ACTION Control:
IF NOT bRUN THEN
				lrGearRatio:=-ABS(lrLifterStopDosePosition-lrLifterStartDosePosition+0.000000000001)
							/(*---------------------------------------------------------------------*)
							((BOOL_TO_INT(bLiftSynchroPh1)*lrDosePhase1Volume)
							+(BOOL_TO_INT(bLiftSynchroPh2)*(lrDoseVolume-lrDosePhase2Volume-lrDosePhase1Volume))
							+((BOOL_TO_INT(bLiftSynchroPh3)*(lrDoseVolume-lrDosePhase1Volume)))
							+ 0.000000000001); 					
	drugafaza:=(lrDoseVolume-lrDosePhase2Volume-lrDosePhase1Volume);						
	trzeciafaza:=(lrDoseVolume-lrDosePhase2Volume);
	calosc:=(*---------------------------------------------------------------------*)
							((BOOL_TO_INT(bLiftSynchroPh1)*lrDosePhase1Volume)
							+(BOOL_TO_INT(bLiftSynchroPh2)*(lrDoseVolume-lrDosePhase2Volume-lrDosePhase1Volume))
							+((BOOL_TO_INT(bLiftSynchroPh3)*lrDosePhase2Volume))
							+ 0.000000000001);
END_IF
	



	(** TIMERY**)
	tonDoseValveOpenTimeAcc(	IN:= eRunningState = E_DispencerState.eDosingPh1, 											PT:= LREAL_TO_TIME(lrDoseValveOpenTimeAcc));   		// [1] Przyśpieszenie otwarcia zaworu tłoczenia [ms]
	tonDoseValveCloseTimeDec(	IN:= (eRunningState=E_DispencerState.eDosingPh3 AND NOT bDoseSucking) OR
									 (eRunningState=E_DispencerState.eDoseSucking AND mcDispencerMoveAbsolute1.Done),		PT:= LREAL_TO_TIME(lrDoseValveCloseTimeDec));  		// [2] Opóźnienie zamknięcia zaworu tłoczenia [ms]
	tonSuckValveOpenTimeDelay(	IN:= eRunningState = E_DispencerState.eGoingUp,											PT:= LREAL_TO_TIME(lrSuckValveOpenTimeDelay));		// [3] Opóżnienie rozpoczęcia ssania po tłoczeniu [ms]
	tonSuckValveCloseTimeDelay(	IN:= (eRunningState = E_DispencerState.eSucking OR 
										eRunningState = E_DispencerState.eDosingDone											
																	) AND
										 mcDispencerMoveAbsolute1.Done, 												PT:= LREAL_TO_TIME(lrSuckValveCloseTimeDelay)); 	// [4] Opóżnienie zamknięcia zaworu ssącego [ms]
	tonDoseSuckingTimeDelay(	IN:= eRunningState = E_DispencerState.eDoseSucking,										PT:= LREAL_TO_TIME(lrDoseSuckingTimeDelay));    	// [6] [Podsysanie] Opóźnienie podsysania [ms]

	//Opóźnienie potwierdzenia wykonania dozy
	(*tonDosingDoneDelay(IN:=(eRunningState=E_DispencerState.eDosingDone OR eRunningState=E_DispencerState.eSucking)AND
							mcDispencerMoveAbsolute1.Done AND tonSuckValveCloseTimeDelay.Q 				
							, PT:=UDINT_TO_TIME(nDosingDoneDelayTime));*)
	tonPrepareToAborting(IN:=bPrepareToAborting, PT:=T#1S);
	//Opóźnienie potwierdzenia wykonania dozy Zmiana 20200820
	tonDosingDoneDelay(IN:=(eRunningState=E_DispencerState.eDosingDone OR eRunningState=E_DispencerState.eSucking)				
							, PT:=UDINT_TO_TIME(nDosingDoneDelayTime));
							
	tonDelayServoOn(IN:=(eState = E_Station.ePreparingToReady), PT:=T#7S); ////bylo 3 Nowe XTS bylo 1200ms						
	tonDelayEnable(IN:=	bEnable, PT:=T#5S);			
	(*Synchronizacja tylko jedna zaznaczona*)
	(*Zabezpieczenie przed zalaczeniem trzech*)
(*	rtLiftSynchroPh3(CLK:=bLiftSynchroPh3,Q=>);rtLiftSynchroPh2(CLK:=bLiftSynchroPh2,Q=>);rtLiftSynchroPh1(CLK:=bLiftSynchroPh1,Q=>);
	IF rtLiftSynchroPh1.Q THEN	bLiftSynchroPh2:=FALSE;	bLiftSynchroPh3:=FALSE; END_IF
	IF rtLiftSynchroPh2.Q THEN	bLiftSynchroPh1:=FALSE;	bLiftSynchroPh3:=FALSE; END_IF
	IF rtLiftSynchroPh3.Q THEN	bLiftSynchroPh1:=FALSE;	bLiftSynchroPh2:=FALSE; END_IF 
	IF bLiftSynchroPh1 THEN	bLiftSynchroPh2:=FALSE;	bLiftSynchroPh3:=FALSE;
	ELSIF bLiftSynchroPh2 THEN	bLiftSynchroPh1:=FALSE;	bLiftSynchroPh3:=FALSE;
	ELSIF bLiftSynchroPh3 THEN	bLiftSynchroPh1:=FALSE;	bLiftSynchroPh2:=FALSE;
	ELSIF NOT bLiftSynchroPh1  AND NOT bLiftSynchroPh2 AND NOT bLiftSynchroPh3 THEN	bLiftSynchroPh1:=TRUE;	bLiftSynchroPh2:=FALSE;	bLiftSynchroPh3:=FALSE; END_IF
	(*Koniec Zabezpieczenie przed zalaczeniem trzech*)
*)
	
	//	100					300			250
	IF lrDosePhase1Volume>lrDoseVolume-lrDosePhase2Volume THEN
		lrDosePhase1Volume:=lrDoseVolume-lrDosePhase2Volume;
	END_IF
	// 200					300			200
	IF lrDosePhase2Volume>lrDoseVolume-lrDosePhase1Volume THEN
		lrDosePhase2Volume:=lrDoseVolume-lrDosePhase1Volume;
	END_IF
	
	IF  eState=E_Station.eReady OR eRunningState=E_DispencerState.eDosingDone OR eRunningState=E_DispencerState.eGoingUp THEN
//	IF  (eState>E_Station.eError AND eState<=E_Station.eReady) OR eRunningState=E_DispencerState.eDosingDone OR eRunningState=E_DispencerState.eGoingUp THEN
		IF (DispencerLifterAxisRef.NcToPlc.ActPos  >= lrDropCatcherHeightCV+(lrDropCatcherOpenDistance-5)) AND lrDropCatcherHeightCV>1 AND NOT bHoming AND NOT bHeightSet THEN
			bDropCatcherActuator:=TRUE;
		ELSE
			bDropCatcherActuator:=FALSE;
		END_IF
	END_IF
							
							
	//Zbocza 
	rtDosingPh1(CLK:=eRunningState=E_DispencerState.eDosingPh1,Q=>);
	rtDosingPh2(CLK:=eRunningState=E_DispencerState.eDosingPh2,Q=>);
	rtDosingPh3(CLK:=eRunningState=E_DispencerState.eDosingPh3,Q=>);
	rtGoingUp(CLK:=eRunningState=E_DispencerState.eGoingUp,Q=>);
	rtPreparingToDose(CLK:=eRunningState=E_DispencerState.ePreparingToDose,Q=>);	
	
	(*****Wyłączenie enable*****)
	IF NOT bEnable THEN
		IF eState <> E_Station.eDisabled AND eState <> E_Station.ePreparingToDisable THEN
				eState 				:= E_Station.ePreparingToDisable; 
				bCycleDone			:= FALSE;
		END_IF	
	END_IF

	(*****Estop*****)
	IF (NOT bEstop AND bInLimitSwitchSensor) OR (NOT bEStopButtonsAndDoors AND NOT bInLimitSwitchSensor) THEN	
		IF eState <> E_Station.eAborted AND eState <> E_Station.eAborting AND eState <> E_Station.eDisabled THEN
				eState 				:= E_Station.eAborting; 
		END_IF
	END_IF

	
	CASE eState OF
	/////////////////////////////	
		E_Station.eDisabled: 					// Stan nieaktywnosci (Stacja wyłączona) 
		
			IF bEnable AND tonDelayEnable.Q THEN
				eState 				:= E_Station.ePreparingToReady; 
			END_IF 
			
    /////////////////////////////	    
		E_Station.eAborted: 					// Stan bezpiecznego zatrzymania (po Abortingu) 

			IF bEStop THEN
				eState 				:= E_Station.ePreparingToReady;
			END_IF
			
	/////////////////////////////	
		E_Station.eAborting:                 	// Stan bezpiecznego zatrzymywania (po EStopie)
		
			mcDispencerPower.Override			:= 100;
			mcDispencerStop.Execute				:= NOT bStopped AND bDispencerServoPower; //Nowe XTS
			mcDispencerMoveAbsolute1.Execute	:= FALSE;
			mcDispencerMoveAbsolute2.Execute	:= FALSE;
			mcDispencerManualMove.JogBackwards	:= FALSE;
			mcDispencerManualMove.JogForward	:= FALSE;			
			
			IF bDispencerWithLifter THEN (*n*)
				mcLifterPower.Override				:= 100;
				mcLifterStop.Execute				:= NOT bStopped AND bLifterServoPower; //Nowe XTS
				mcLifterMoveAbsolute.Execute		:= FALSE;	
				mcLifterManualMove.JogBackwards		:= FALSE;
				mcLifterManualMove.JogForward		:= FALSE;
				bHeightSetNotDone 					:= FALSE; //Zmiana 2021-02-19
			END_IF	
											(*n*)					//Zmiana XTS
			IF ((mcLifterStop.Done OR NOT bDispencerWithLifter OR NOT bLifterServoPower) AND (mcDispencerStop.Done OR NOT bDispencerServoPower)) OR bStopped THEN
				
				mcDispencerStop.Execute			:=	FALSE;
				bDispencerServoPower			:=	FALSE;
				
				mcLifterStop.Execute			:=	FALSE;
				bLifterServoPower				:=	FALSE;
				
				bStopped						:=	FALSE;
				eState							:=	E_Station.eAborted; 
				eRunningState					:=	E_DispencerState.eReady;
			END_IF	
					
	/////////////////////////////			
		E_Station.eError:                 	 	// Stan błędu 	
			
			IF bReset OR tofReset.Q THEN
				eState 				:= E_Station.eResetting;
				eRunningState		:= E_DispencerState.eReady;
			ELSE
				mcLifterSoftReset	(Execute:=FALSE,Axis:=DispencerLifterAxisRef);
				mcDispencerSoftReset(Execute:=FALSE,Axis:=DispencerAxisRef);
			END_IF
			
	/////////////////////////////
		E_Station.eResetting:					// Stan resetowania bledu (po Errorze)
			
			//Procedura obsługi resetu w zależności od błędu
			CASE nErrorNr-iStationIndex OF
		
				//Error 2 - BŁĄD SERWA DOZOWNIKA
				1:	
					mcDispencerSoftReset(Execute:=TRUE,Axis:=DispencerAxisRef);
					IF mcLifterGearIn.InGear THEN
						mcLifterGearIn.Enable:=FALSE;
						mcLifterGearOut.Execute := TRUE;
					END_IF
					IF mcLifterGearOut.Done THEN
						mcLifterGearOut.Execute := FALSE;
					END_IF
					IF NOT mcLifterGearIn.InGear AND NOT mcLifterGearOut.Execute THEN
					
						IF NOT fbDispencerHardReset.Busy AND NOT mcDispencerSoftReset.Busy AND mcDispencerPower.Status AND NOT DispencerAxisRef.Status.Error THEN
								mcDispencerSoftReset(Execute:=FALSE,Axis:=DispencerAxisRef);
								nErrorNr:=0;
								nDispencerServoErrorNr:=0;
								bError := FALSE;
								sErrorDescription:='';	
				
						ELSIF NOT fbDispencerHardReset.Busy AND NOT mcDispencerSoftReset.Busy AND NOT mcDispencerPower.Status AND NOT DispencerAxisRef.Status.Error THEN
								nErrorNr:=0;
								nDispencerServoErrorNr:=0;
								bError := FALSE;
								sErrorDescription:='';
						END_IF
						IF fbDispencerHardReset.Error OR mcDispencerSoftReset.Error THEN
							mcDispencerSoftReset(Execute:=FALSE,Axis:=DispencerAxisRef);
						END_IF
						
					END_IF

				//Error 2, Error 4 - BŁĄD SERWA PODNOSZENIA DOZOWNIKA
				2:	
					mcLifterGearIn.Enable:=FALSE;
					mcLifterGearOut.Execute:=FALSE;
					//fbLifterHardReset(Execute:=NOT mcLifterMoveAbsolute.Execute,Axis:=DispencerLifterAxisRef);
					mcLifterSoftReset(Execute:=NOT mcLifterMoveAbsolute.Execute,Axis:=DispencerLifterAxisRef);
					IF NOT fbLifterHardReset.Busy AND NOT mcLifterSoftReset.Busy AND mcLifterPower.Status AND NOT DispencerLifterAxisRef.Status.Error THEN
						//fbLifterHardReset(Execute:=FALSE,Axis:=DispencerLifterAxisRef);
						mcLifterSoftReset(Execute:=FALSE,Axis:=DispencerLifterAxisRef);
						mcLifterMoveAbsolute.Execute:=TRUE;
						mcLifterMoveAbsolute.Position:=lrLifterReadyPosition;
						mcLifterPower.Override:=100; 
						IF mcLifterMoveAbsolute.Done THEN
							bDropCatcherActuator:=TRUE;
							mcLifterPower.Override:=100; 
							mcLifterMoveAbsolute.Execute:=FALSE;
							nErrorNr:=0;
							nLifterServoErrorNr:=0;
							bError := FALSE;
							sErrorDescription:='';	
						END_IF 
					ELSIF NOT fbLifterHardReset.Busy AND NOT mcLifterSoftReset.Busy AND NOT mcLifterPower.Status AND NOT DispencerLifterAxisRef.Status.Error THEN		
						//fbLifterHardReset(Execute:=FALSE,Axis:=DispencerLifterAxisRef);
						mcLifterSoftReset(Execute:=FALSE,Axis:=DispencerLifterAxisRef);
						nErrorNr:=0;
						nLifterServoErrorNr:=0;
						bError := FALSE;
						sErrorDescription:='';	
					END_IF
					IF fbLifterHardReset.Error OR mcLifterSoftReset.Error THEN
						//fbLifterHardReset(Execute:=FALSE,Axis:=DispencerLifterAxisRef);
						mcLifterSoftReset(Execute:=FALSE,Axis:=DispencerLifterAxisRef);
					END_IF	

				// inny numer błędu
				ELSE
					bSuckingValveActuator:=FALSE;
					bDosingValveActuator:=FALSE;
					IF bDispencerWithLifter THEN
						mcLifterSoftReset(Execute:=FALSE,Axis:=DispencerLifterAxisRef);
						mcLifterPower.Override				:=	100; 
						mcLifterMoveAbsolute.Acceleration	:=	lrLifterAcceleration;
						mcLifterMoveAbsolute.Velocity		:=	lrLifterVelocity;
						mcLifterMoveAbsolute.Position		:=	lrLifterReadyPosition;
						mcLifterMoveAbsolute.Execute		:=	bLifterServoPower; 
						IF mcLifterMoveAbsolute.Done OR NOT bLifterServoPower THEN 
							bDropCatcherActuator:=TRUE;
							mcLifterPower.Override:=100; 
							mcLifterMoveAbsolute.Execute:=FALSE;
							nErrorNr:=0;
							nLifterServoErrorNr:=0;
							bError := FALSE;
							sErrorDescription:='';	
						END_IF
					ELSE
						bError := FALSE;
					END_IF 

			END_CASE	
			
			IF NOT bError THEN
				nErrorNr 			:=	0;
   				sErrorDescription 	:=	'';
	
				eState 				:=	E_Station.ePreparingToReady;
			ELSE
				eState 				:=	E_Station.eError;
			END_IF
        
	/////////////////////////////
		E_Station.eManualMovement:     			// Stan ruchów manualnych  
       
			ManualMovements();
			//Wyjście z trybu serwisowego
			IF NOT bManualMovement AND bInLimitSwitchSensor  AND NOT bChangeover THEN
				mcDispencerPower.Override			:=	100;		
				bSuckingValveActuator				:=	FALSE;
				bDosingValveActuator				:=	FALSE;
				mcDispencerMoveAbsolute1.Execute	:=	FALSE;
			
				IF bDispencerWithLifter THEN
					IF lrLifterActualPosition < lrLifterReadyPosition + 1 THEN
						mcLifterMoveAbsolute.Execute		:= TRUE;
						mcLifterMoveAbsolute.Acceleration	:= lrLifterAcceleration;
						mcLifterMoveAbsolute.Velocity		:= lrLifterVelocity;
						mcLifterMoveAbsolute.Position		:= lrLifterReadyPosition;
					END_IF
				END_IF
				
				IF NOT bDispencerWithLifter OR mcLifterMoveAbsolute.Done OR lrLifterActualPosition >= lrLifterReadyPosition THEN
					mcDispencerMoveAbsolute1.Execute:=FALSE;
					mcLifterMoveAbsolute.Execute:=FALSE;
					eState 							:= E_Station.eReady;
				END_IF
			END_IF

	/////////////////////////////
		E_Station.eHoming:						// Stan bazowania 

			Homing();
			IF NOT bHoming AND NOT bHeightSet THEN
			   eState:=E_Station.ePreparingToReady;
			   	mcLifterManualMove.JogForward		:= FALSE;
				mcLifterManualMove.JogBackwards		:= FALSE;
			END_IF			
			
	/////////////////////////////
		E_Station.eHomingDone:                  // Stan wykonania bazowania 
		
			bHomingDone							:=	TRUE;
			IF NOT bHoming AND NOT bHeightSet THEN
				
			   eState:=E_Station.eReady;
			END_IF
			
	/////////////////////////////
		E_Station.ePreparingToReady:            // Stan przygotowywania do gotowosci (zawsze przed Ready)  

		
			IF tonDelayServoOn.Q THEN
				bDispencerServoPower		:= TRUE;		
				bLifterServoPower			:= TRUE;//bDispencerWithLifter	; (*n*) //ZMIANA XTS
			END_IF	
		
			mcDispencerPower.Override	:= 100;
			bDosingValveActuator		:= FALSE;
			bSuckingValveActuator		:= FALSE;
			bManualDosingValve			:= FALSE;
			bManualSuckingValve			:= FALSE;
			bServiceBrakeOff			:= FALSE;

			mcLifterMoveAbsolute.Execute := FALSE;

			mcDispencerMoveAbsolute1.Execute := FALSE;
			mcDispencerMoveAbsolute2.Execute := FALSE;
			mcDispencerMoveAbsolute3.Execute := FALSE;
				(*n*)
			IF (mcLifterPower.Status OR NOT bDispencerWithLifter) AND mcDispencerPower.Status THEN
											(*n*)
				IF NOT bHeightSetNotDone AND bDispencerWithLifter THEN
					
					IF mcLifterGearIn.InGear THEN
						mcLifterGearIn.Enable := FALSE;
						mcLifterGearOut.Execute := TRUE;
					ELSIF mcLifterGearIn.Enable AND mcLifterGearOut.Done THEN 
						mcLifterGearOut.Execute := FALSE;
					ELSE
						mcLifterPower.Override:=100;
						mcLifterMoveAbsolute.Velocity:=1000;
						mcLifterMoveAbsolute.Execute:= TRUE;
						mcLifterMoveAbsolute.Position:=lrLifterReadyPosition;
						IF bChangeover THEN
							mcLifterMoveAbsolute.Position:=lrMaxPosition;
						END_IF
						IF mcLifterMoveAbsolute.Done THEN
							mcLifterMoveAbsolute.Execute:=FALSE;
							eState:=E_Station.eReady;
							eRunningState:=E_DispencerState.eReady;
						END_IF
					END_IF
					
				ELSE
					bHeightSetNotDone := FALSE;
					eState:=E_Station.eReady;
					eRunningState:=E_DispencerState.eReady;
				END_IF	
			END_IF
         	IF bIgnoreError THEN
				eState:=E_Station.eReady;
				eRunningState:=E_DispencerState.eReady;
			END_IF


	
				
	/////////////////////////////
		E_Station.ePreparingToDisable:          // Stan przygotowywania do nieaktywnosci (po wyłączeniu Enable) 
  			bDropCatcherActuator:=FALSE; //Zmiana 29072019
			mcDispencerPower.Override:=100;
			mcLifterPower.Override:=100;
			IF bPreparingToDisable THEN
				mcLifterStop.Execute:=FALSE;
				mcLifterMoveAbsolute.Execute:= NOT mcLifterStop.Execute AND NOT  mcLifterStop.DONE;
				mcLifterMoveAbsolute.Position:=lrMaxPosition;
				mcLifterMoveAbsolute.Acceleration:=lrLifterAcceleration;
				mcLifterMoveAbsolute.Deceleration:=lrLifterDeceleration;
				mcLifterMoveAbsolute.Velocity:=lrLifterVelocity;
				IF mcLifterMoveAbsolute.Done THEN
					mcLifterMoveAbsolute.Execute:=FALSE;
					eState:=E_Station.eDisabled;
					bPreparingToDisable := FALSE;
					bDispencerServoPower:=FALSE;
					bLifterServoPower:=FALSE;
				END_IF
			ELSE
				mcDispencerStop.Execute:=NOT mcDispencerMoveAbsolute1.Execute AND NOT mcDispencerMoveAbsolute2.Execute AND NOT mcDispencerMoveAbsolute3.Execute;
				mcDispencerMoveAbsolute1.Execute:=FALSE;
				mcDispencerMoveAbsolute2.Execute:=FALSE;
				mcDispencerMoveAbsolute3.Execute:=FALSE;
		
				IF 	mcDispencerStop.Done  THEN
								
					IF bDispencerWithLifter AND DispencerLifterAxisRef.NcToPlc.CoupleState<3 THEN
						mcLifterGearOut.Execute:=FALSE;
						mcLifterGearIn.Enable:=FALSE;			
						mcLifterStop.Execute:=NOT mcLifterMoveAbsolute.Execute;
						mcLifterMoveAbsolute.Execute:=FALSE;
						mcLifterStop.Execute:=TRUE;
					ELSIF  bDispencerWithLifter AND DispencerLifterAxisRef.NcToPlc.CoupleState=3 THEN
						mcLifterGearIn.Enable:=FALSE;
						mcLifterGearOut.Execute:=TRUE;
					END_IF
		
					IF bEstop AND (bDispencerWithLifter AND DispencerLifterAxisRef.NcToPlc.CoupleState<3) THEN
						bPreparingToDisable:=TRUE;
						bSuckingValveActuator:=FALSE;
						bDosingValveActuator:=FALSE;;
					
					ELSIF (NOT bDispencerWithLifter OR mcLifterStop.Done) AND mcDispencerStop.Done THEN
						bDispencerServoPower:=FALSE;
						bDropCatcherActuator:=FALSE;
						IF bDispencerWithLifter THEN
							bLifterServoPower:=FALSE;
							mcLifterGearOut.Execute:=FALSE;
							mcLifterStop.Execute:=FALSE;
						END_IF
						mcDispencerStop.Execute:=FALSE;
						eState:=E_Station.eDisabled;
						mcDispencerStop.Execute:=FALSE;
						
						bSuckingValveActuator:=FALSE;
						bDosingValveActuator:=FALSE;
					END_IF
				END_IF
			END_IF
			
	/////////////////////////////
		E_Station.eReady:						// Stan gotowosci 

			IF bRun AND NOT bCycleDone AND NOT bCycleNotDone THEN
				eState 				:= E_Station.eStarting; 
			END_IF
			IF bHoming OR bHeightSet THEN
				eState 				:= E_Station.eHoming; 
			END_IF
			IF bManualMovement OR NOT bInLimitSwitchSensor OR bChangeover THEN //Przejscie do serwisu jak nie ma na czujniku
				IF NOT bInLimitSwitchSensor THEN
					bLifterServoPower		:=	FALSE;
				END_IF
				//Jeśli przejście w tryb ruchów manualnych przepisz wszystkie stany siłowników sterowanych przez moduł
				//aby zapobiec ewentualnym kolizjom po wejściu w tryb serwisowy
				bManualDosingValve			:=	bDosingValveActuator;
				bManualSuckingValve			:=	bSuckingValveActuator;
				bManualDropCatcherForward	:=	bDropCatcherActuator;
				mcDispencerStop.Execute		:=	FALSE;
				//eState 						:=	E_Station.eManualMovement; 
			
				// Dodanie zmieny narzędzia, zamiast wyłączenia stacja jedzie do góry i będzie możliwość
				// tych samych funkcji co w trybie serwisowy, przeciągania itp
				IF bChangeover THEN
					IF bDispencerWithLifter THEN
						IF lrLifterActualPosition < lrMaxPosition + 1 THEN
							mcLifterMoveAbsolute.Execute		:= TRUE;
							mcLifterMoveAbsolute.Acceleration	:= lrLifterAcceleration/3;
							mcLifterMoveAbsolute.Velocity		:= lrLifterVelocity/3;
							mcLifterMoveAbsolute.Position		:= lrMaxPosition;
						END_IF
					END_IF
					
					IF NOT bDispencerWithLifter OR mcLifterMoveAbsolute.Done OR lrLifterActualPosition >= lrMaxPosition  THEN
						mcDispencerMoveAbsolute1.Execute	:=FALSE;
						mcLifterMoveAbsolute.Execute		:=FALSE;
						eState 						:=	E_Station.eManualMovement; 
					END_IF
				ELSE
					eState 						:=	E_Station.eManualMovement; 
				END_IF	
			
			END_IF
			IF NOT bRun THEN
				bCycleDone 					:= FALSE;
				bCycleNotDone 				:= FALSE;	
			END_IF
			
			bStopped						:= FALSE;
			mcLifterStop.Execute			:= FALSE;
			mcDispencerStop.Execute			:= FALSE;
			
	/////////////////////////////
		E_Station.eStopping:					// Stan zatrzymywania 
			eRunningState:=E_DispencerState.eReady;//zmiana 20200820
			Running();
			
			mcDispencerPower.Override:=100;
			mcLifterPower.Override:=100;
			mcDispencerStop.Execute:= NOT mcDispencerMoveAbsolute1.Execute AND NOT mcDispencerMoveAbsolute2.Execute AND NOT mcDispencerMoveAbsolute3.Execute AND NOT mcDispencerStop.CommandAborted;
			mcDispencerMoveAbsolute1.Execute:=FALSE;
			mcDispencerMoveAbsolute2.Execute:=FALSE;
			mcDispencerMoveAbsolute3.Execute:=FALSE;
			IF mcDispencerStop.Done THEN
				bDosingValveActuator:=FALSE;
				bSuckingValveActuator:=FALSE;
				IF bDispencerWithLifter THEN
					mcLifterMoveAbsolute.Execute:=FALSE;
					mcLifterMoveAbsolute.BufferMode:=MC_Aborting;
					mcLifterGearIn.Enable:=FALSE;
					mcLifterGearOut.Execute:=TRUE;
					IF mcLifterGearOut.Done THEN; 
						
						mcLifterMoveAbsolute.Execute:=bStopped;
						//mcDispencerStop.Execute:=FALSE;
						IF mcLifterStop.DONE THEN
							bStopped:=TRUE;
						END_IF
						mcLifterStop.Execute:=NOT bStopped;
						
						mcLifterMoveAbsolute.Acceleration:=lrLifterAcceleration;
						mcLifterMoveAbsolute.Deceleration:=lrLifterDeceleration;
						mcLifterMoveAbsolute.Velocity:=lrLifterVelocity;
						mcLifterMoveAbsolute.Position:=lrLifterReadyPosition;
						
						IF mcLifterMoveAbsolute.Done AND bStopped THEN
							//mcLifterMoveAbsolute.Execute:=FALSE;
							//mcLifterMoveAbsolute.BufferMode:=MC_Aborting;
							eState:=E_Station.eReady;
							bStopped:=FALSE;
							bDropCatcherActuator:=TRUE;
							mcDispencerStop.Execute:=FALSE;
							mcLifterMoveAbsolute.Execute:=FALSE;
							mcLifterGearOut.Execute:=FALSE;
						END_IF
					END_IF
				ELSE
					mcDispencerStop.Execute:=FALSE;
					eState:=E_Station.eReady;
				END_IF
			END_IF
	
			IF mcLifterMoveAbsolute.Error THEN
				mcLifterMoveAbsolute.Execute:=FALSE;
			END_IF
			
	/////////////////////////////
		E_Station.eStarting:                  	// Stan uruchamiania (po Ready)
		
			eState					 := E_Station.eRunning; 
			
	/////////////////////////////
		E_Station.eRunning:               		// Stan wykonywania cyklu (po Startingu), w tym stanie osobny
 
			Running();
			IF NOT bRun THEN					(*Przerywanie cyklu*)
				eState 				 := E_Station.eStopping;	
				bCountTestDoz1:=bCountTestDoz1+1;
			END_IF
			IF bCycleDone OR bCycleNotDone THEN (*Cykl zakończony*)
				eState 				 := E_Station.eReady;
				eRunningState		 := E_DispencerState.eReady;//zmiana 20200820
				bCountTestDoz2:=bCountTestDoz2+1;
			END_IF	
			
			
	/////////////////////////////		
	END_CASE
END_ACTION

ACTION DispencerControlBlocks:
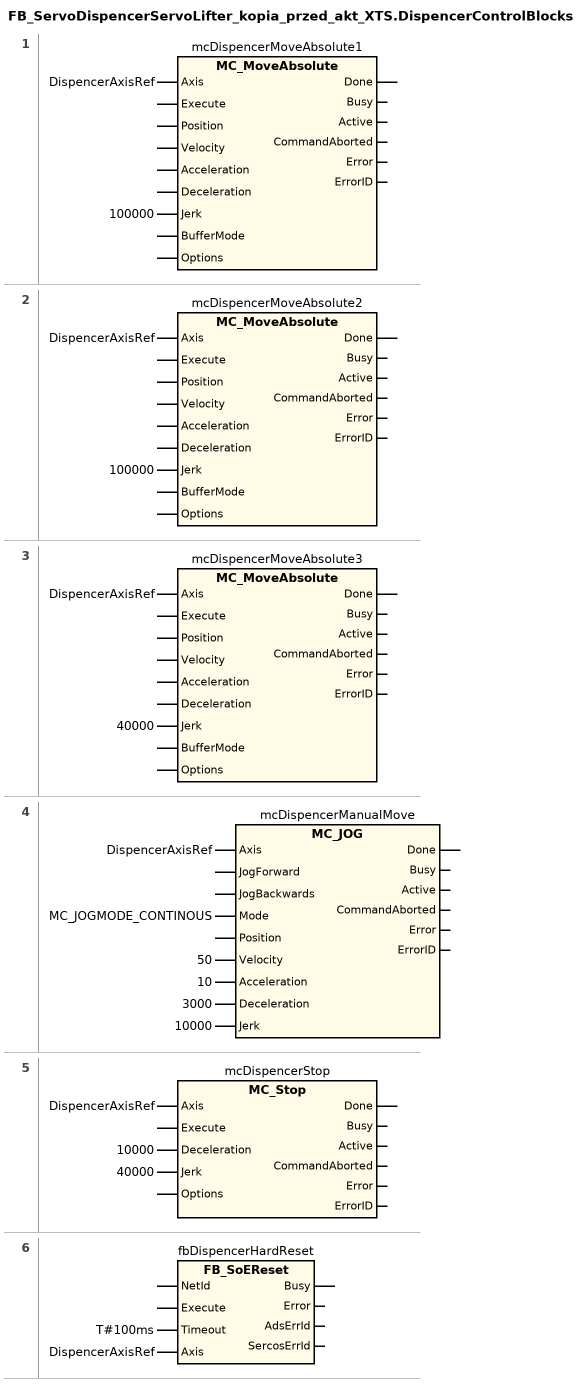
// NETWORK 1
mcDispencerMoveAbsolute1(Axis := DispencerAxisRef, Jerk := 100000); // MC_MoveAbsolute

// NETWORK 2
mcDispencerMoveAbsolute2(Axis := DispencerAxisRef, Jerk := 100000); // MC_MoveAbsolute

// NETWORK 3
mcDispencerMoveAbsolute3(Axis := DispencerAxisRef, Jerk := 40000); // MC_MoveAbsolute

// NETWORK 4
mcDispencerManualMove(
    Axis := DispencerAxisRef,
    Mode := MC_JOGMODE_CONTINOUS,
    Velocity := 50,
    Acceleration := 10,
    Deceleration := 3000,
    Jerk := 10000); // MC_JOG

// NETWORK 5
mcDispencerStop(Axis := DispencerAxisRef, Deceleration := 10000, Jerk := 40000); // MC_Stop

// NETWORK 6
fbDispencerHardReset(Timeout := T#100ms, Axis := DispencerAxisRef); // FB_SoEReset

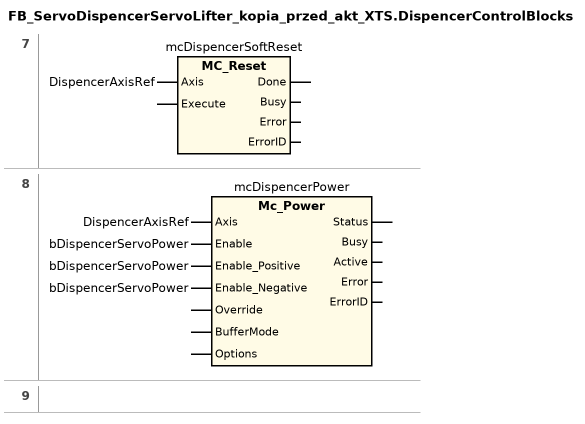
// NETWORK 7
mcDispencerSoftReset(Axis := DispencerAxisRef); // MC_Reset

// NETWORK 8
mcDispencerPower(
    Axis := DispencerAxisRef,
    Enable := bDispencerServoPower,
    Enable_Positive := bDispencerServoPower,
    Enable_Negative := bDispencerServoPower); // Mc_Power

// NETWORK 9
END_ACTION

ACTION ErrorHandling:
//OBSŁUGA BŁĘDÓW DOZOWNIKA Z PODNOŚNIKIEM EPCO

DispencerAxisRef.ReadStatus();

(**Błąd tylko podczas cyklu*)
bErrorOnlyIfCycleOn :=	(eRunningState=E_DispencerState.ePreparingToDose) OR 
						(eRunningState=E_DispencerState.eDosingPh1) OR 
						(eRunningState=E_DispencerState.eDosingPh2) OR 
						(eRunningState=E_DispencerState.eDosingPh3) OR 
						(eRunningState=E_DispencerState.eDosingDone) OR 
						(eRunningState=E_DispencerState.ePulling) OR 
						(eRunningState=E_DispencerState.eSucking) OR 
						(eRunningState=E_DispencerState.eGoingUp) OR 
						(eRunningState=E_DispencerState.eAborting) OR
						(eRunningState=E_DispencerState.eDoseSucking) OR
						(eRunningState=E_DispencerState.eDoseSuckingDone); 
tonEstopDelay			(IN:=bEstop,	PT:=T#2S); //Opóżnienie po EStopie w celu blokoady błędów, powietrze jest później niż Estop a sygnał z czujnika nie pokazuje braku powietrza bo jest odcinany za tym
						
//**********************LISTA BŁĘDÓW******************************
bStateError:= (eState=E_Station.eError) OR (eState=E_Station.eResetting) OR bIgnoreError;

IF bEnable THEN
	
	//Error 1 - BŁĄD SERWA DOZOWNIKA 
	IF DispencerAxisRef.Status.Error AND NOT bStateError THEN
		bManualPullingLatch:=FALSE;
		mcDispencerPower.Override:=100;
		bError := TRUE;
		mcDispencerMoveAbsolute1.Execute:=FALSE;
		mcDispencerMoveAbsolute2.Execute:=FALSE;
		mcDispencerMoveAbsolute3.Execute:=FALSE;
		nErrorNr:=1;
		nErrorNr := nErrorNr+iStationIndex;
		nDispencerServoErrorNr:=DispencerAxisRef.Status.ErrorID;
		bSuckingValveActuator:=FALSE;
		bDosingValveActuator:=FALSE;
		sErrorDescription:='Błąd napędu tłoka - upewnij się że został dobrze złożony. Błąd NC:';
		sErrorDescription2:=F_AxErrMsg(nDispencerServoErrorNr);
	END_IF

	//Error 2 - BŁĄD SERWA PODNOSNIKA DOZOWNIKA
	IF bDispencerWithLifter AND (DispencerLifterAxisRef.Status.Error OR mcLifterPower.Error) AND NOT bStateError THEN
		bManualPullingLatch:=FALSE;
		bSuckingValveActuator:=FALSE;
		bDosingValveActuator:=FALSE;
		mcDispencerPower.Override:=100;
		mcLifterGearIn.Enable:=FALSE;
		mcLifterGearOut.Execute:=TRUE;
		mcLifterPower.Override:=100;
		mcLifterMoveAbsolute.Execute:=FALSE;
		bError := TRUE;
		nErrorNr:=2;
		nErrorNr := nErrorNr+iStationIndex;
		nLifterServoErrorNr:=DispencerLifterAxisRef.Status.ErrorID;
		sErrorDescription:='Błąd napędu podnośnika. Błąd NC:';
		sErrorDescription2:=F_AxErrMsg(nLifterServoErrorNr);	
	END_IF;
		
	//Error 3 - Nastawa dozy większa niż objętość robocza dozownika
	IF bRun AND eState=E_Station.eReady AND lrDoseVolume>lrRatedDose AND NOT bStateError THEN
		bManualPullingLatch:=FALSE;
		bSuckingValveActuator:=FALSE;
		bDosingValveActuator:=FALSE;
		mcDispencerPower.Override:=100;
		bError := TRUE;
		nErrorNr:=3;
		nErrorNr := nErrorNr+iStationIndex;
		sErrorDescription:='Nastawa dozy powyżej maksymalnej wartości - zmniejsz ilość dozy';
		sErrorDescription2:=LREAL_TO_STRING(lrDoseVolume);
	END_IF
	
	//Error 4 - Nastawa dozy mniejsza niż objętość robocza dozownika
	IF bRun AND eState=E_Station.eReady AND lrDoseVolume<0 AND NOT bStateError THEN
		bManualPullingLatch:=FALSE;
		bSuckingValveActuator:=FALSE;
		bDosingValveActuator:=FALSE;
		mcDispencerPower.Override:=100;
		bError := TRUE;
		nErrorNr:=4;
		nErrorNr := nErrorNr+iStationIndex;
		sErrorDescription:='Nastawa dozy poniżej minimalnej wartość - zwiększ ilość dozy';
		sErrorDescription2:=LREAL_TO_STRING(lrDoseVolume);
	END_IF
	
	//Error 5 - Blokada zaworu ssania przy zamykaniu																					  (*tylko podczas cyklu*)
	tonSuckingValveCloseError(IN:=NOT bSuckingValveClosedSensor AND NOT bSuckingValveActuator AND NOT bStateError AND bErrorOnlyIfCycleOn, PT:=T#1S);
	IF NOT bIgnoreError AND tonSuckingValveCloseError.Q AND NOT bStateError THEN
		bError := TRUE;
		nErrorNr:=5;
		nErrorNr := nErrorNr+iStationIndex;
		sErrorDescription:='Zacięcie zaworu zasysania podczas zamykania - sprawdź czujnik';
	END_IF
	
	//Error 6 - Blokada zaworu ssania przy zamykaniu																				(*tylko podczas cyklu*)
	tonSuckingValveOpenError(IN:=NOT bSuckingValveOpenedSensor AND bSuckingValveActuator AND NOT bStateError AND bErrorOnlyIfCycleOn, PT:=T#1S);
	IF NOT bIgnoreError AND tonSuckingValveOpenError.Q AND NOT bStateError THEN
		bError := TRUE;
		nErrorNr:=6;
		nErrorNr := nErrorNr+iStationIndex;
		sErrorDescription:='Zacięcie zaworu zasysania masy podczas otwierania - sprawdź czujnik';
	END_IF
	
	//Error 7 - Blokada zaworu ssania przy zamykaniu																				(*tylko podczas cyklu*)
	tonDosingValveCloseError(IN:=NOT bDosingValveClosedSensor AND NOT bDosingValveActuator AND NOT bStateError AND bErrorOnlyIfCycleOn, PT:=T#1S);
	IF NOT bIgnoreError AND tonDosingValveCloseError.Q AND NOT bStateError THEN
		bError := TRUE;
		nErrorNr:=7;
		nErrorNr := nErrorNr+iStationIndex;
		sErrorDescription:='Zacięcie zaworu tłoczenia masy podczas zamykania - sprawdź czujnik';
	END_IF
	
	//Error 8 - Blokada zaworu ssania przy zamykaniu																			  (*tylko podczas cyklu*)
	tonDosingValveOpenError(IN:=NOT bDosingValveOpenedSensor AND bDosingValveActuator AND tonEstopDelay.Q AND bStateError AND bErrorOnlyIfCycleOn, PT:=T#1S);
	IF NOT bIgnoreError AND tonDosingValveOpenError.Q AND NOT bStateError THEN
		bError := TRUE;
		nErrorNr:=8;
		nErrorNr := nErrorNr+iStationIndex;
		sErrorDescription:='Zacięcie zaworu tłoczenia masy podczas otwierania - sprawdź czujnik';
	END_IF
	
	//Error 11 - Blokada tacki przy otwieraniu																 (*tylko podczas cyklu*)
	tonDropCatcherOpenError(IN:=NOT bDropCatcherBackSensor AND NOT bDropCatcherActuator AND tonEstopDelay.Q AND NOT bStateError, PT:=T#1S); // było 1S500MS
	IF 	NOT bIgnoreError AND (tonDropCatcherOpenError.Q  OR
        (bRun AND eRunningState>=E_DispencerState.eDosingPh1 AND eRunningState<= E_DispencerState.eDosingPh3 AND NOT bDropCatcherBackSensor))
        AND  NOT bStateError THEN 
		bError := TRUE;
		nErrorNr:=11;
		nErrorNr := nErrorNr+iStationIndex;
		sErrorDescription:='Zacięcie tacki przy zamykaniu - sprawdź czujnik';
		sErrorDescription2:='';
	END_IF
	
	//Error 12 - Próba uruchomienia z zbyt nisko ustawionym chwytakiem (możliwość wylewki w butelce)
	IF NOT bIgnoreError AND 
	(
	(lrLifterActualPosition<(lrDropCatcherHeightCV-40) AND bCatchEnable) OR
	(lrLifterActualPosition<(lrDropCatcherHeightCV-80) AND NOT bCatchEnable) 	
	)
	AND eGlobalState=E_PackMLState.eStarting AND NOT bStateError THEN
		bError := TRUE;
		nErrorNr:=12;
		nErrorNr := nErrorNr+iStationIndex;
		sErrorDescription:='Próba uruchomienia z zbyt niską pozycją wylewki względem chwytaka - zmień pozycję gotowości dozownika lub chwytaka';
		sErrorDescription2:='';
	END_IF	
	
	
ELSE
	bError := FALSE;
END_IF


//Procedura obsługi resetu w zależności od błędu
tofReset(IN:=bReset , PT:=T#3S);
//******************PRZEJŚCIE DO eERROR*****************************

IF bError AND NOT bStateError THEN
	IF eLastState = eRunning THEN
		bCycleNotDone := TRUE;
	END_IF
	eState := E_Station.eError;
END_IF

//****************WYŚWIETLANIE STATUSU BLEDU***********************



(*Wyświetlanie błedu na wyjściu*)
bError;

(*Przepisywanie nazwy stacji*)
sErrorStationName:=sStationName;
END_ACTION

ACTION HardwareHoming:
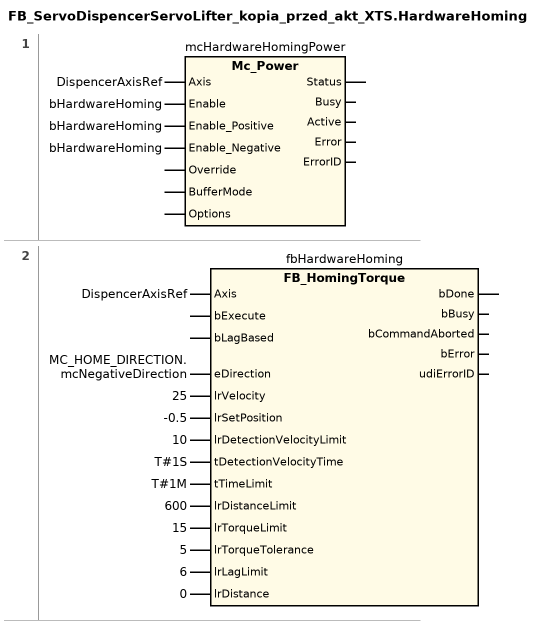
// NETWORK 1
mcHardwareHomingPower(
    Axis := DispencerAxisRef,
    Enable := bHardwareHoming,
    Enable_Positive := bHardwareHoming,
    Enable_Negative := bHardwareHoming); // Mc_Power

// NETWORK 2
fbHardwareHoming(
    Axis := DispencerAxisRef,
    eDirection := MC_HOME_DIRECTION.mcNegativeDirection,
    lrVelocity := 25,
    lrSetPosition := -0.5,
    lrDetectionVelocityLimit := 10,
    tDetectionVelocityTime := T#1S,
    tTimeLimit := T#1M,
    lrDistanceLimit := 600,
    lrTorqueLimit := 15,
    lrTorqueTolerance := 5,
    lrLagLimit := 6,
    lrDistance := 0); // FB_HomingTorque
END_ACTION

ACTION Homing:


bDropCatcherActuator 					:= FALSE;

IF bHoming THEN
	IF bDispencerWithLifter THEN
		mcLifterMoveAbsolute.Velocity		:=100;
		mcLifterMoveAbsolute.Position		:=lrMaxPosition;
		mcLifterMoveAbsolute.Execute		:= TRUE;
		mcLifterPower.Override				:=100;
		IF mcLifterMoveAbsolute.Done THEN
			eState							:= E_Station.eHomingDone;
			mcLifterMoveAbsolute.Execute	:= FALSE;
		END_IF
	ELSE
		IF ABS(DispencerLifterAxisRef.NcToPlc.ActPos-lrMaxPosition)<1 THEN
			eState							:= E_Station.eHomingDone;
		END_IF
	END_IF
ELSIF bHeightSet THEN
	mcLifterManualMove.JogForward:=DispencerLifterAxisRef.NcToPlc.ActPos<=lrLifterReadyPosition AND DispencerLifterAxisRef.NcToPlc.ActPos<=lrMaxPosition;
	mcLifterManualMove.JogBackwards:=DispencerLifterAxisRef.NcToPlc.ActPos>=lrLifterReadyPosition AND DispencerLifterAxisRef.NcToPlc.ActPos>=lrMinPosition;
	IF ABS(DispencerLifterAxisRef.NcToPlc.ActPos-lrLifterReadyPosition)<1 THEN
		mcLifterManualMove.JogForward	:= FALSE;
		mcLifterManualMove.JogBackwards	:= FALSE;
		eState:=E_Station.eHomingDone;
		bHeightSetNotDone					:= TRUE;	
	END_IF
END_IF 
(*
IF NOT bHomingDone THEN
	Lifter_FHPP_CTRL.EnableDrive:=TRUE;
	Lifter_FHPP_CTRL.Stop:=TRUE;
	Lifter_FHPP_CTRL.Halt:=TRUE;
	Lifter_FHPP_CTRL.OPM:=1; 
	IF  Lifter_FHPP_CTRL.Ready THEN
		Lifter_FHPP_CTRL.StartHoming := TRUE;
	END_IF
	IF Lifter_FHPP_CTRL.HomingValid AND tonStartHoming.Q THEN
		Lifter_FHPP_CTRL.StartHoming := FALSE;
		eState:=E_Station.eHomingDone;
	END_IF
ELSE
	lrLifterMaxHeight:=275;
	lrLifterMinHeight:=50;
	Lifter_FHPP_CTRL.JoggingPos:=lrLifterActualPosition<=lrLifterReadyPosition AND lrLifterActualPosition<=lrLifterMaxHeight;
	Lifter_FHPP_CTRL.JoggingNeg:=lrLifterActualPosition>=lrLifterReadyPosition AND lrLifterActualPosition>=lrLifterMinHeight;
	IF ABS(lrLifterActualPosition-lrLifterReadyPosition)<1 THEN
		Lifter_FHPP_CTRL.JoggingPos:=FALSE;
		Lifter_FHPP_CTRL.JoggingNeg:=FALSE;
		eState:=E_Station.eHomingDone;

		
	END_IF		
END_IF*)
END_ACTION

ACTION LifterControlBlocks:
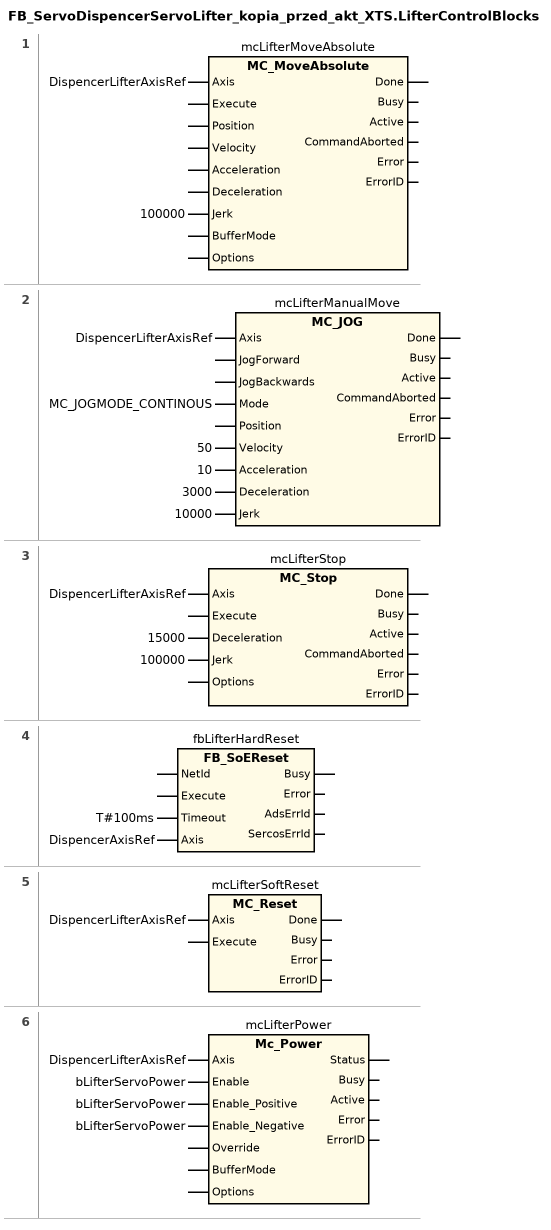
// NETWORK 1
mcLifterMoveAbsolute(Axis := DispencerLifterAxisRef, Jerk := 100000); // MC_MoveAbsolute

// NETWORK 2
mcLifterManualMove(
    Axis := DispencerLifterAxisRef,
    Mode := MC_JOGMODE_CONTINOUS,
    Velocity := 50,
    Acceleration := 10,
    Deceleration := 3000,
    Jerk := 10000); // MC_JOG

// NETWORK 3
mcLifterStop(Axis := DispencerLifterAxisRef, Deceleration := 15000, Jerk := 100000); // MC_Stop

// NETWORK 4
fbLifterHardReset(Timeout := T#100ms, Axis := DispencerAxisRef); // FB_SoEReset

// NETWORK 5
mcLifterSoftReset(Axis := DispencerLifterAxisRef); // MC_Reset

// NETWORK 6
mcLifterPower(
    Axis := DispencerLifterAxisRef,
    Enable := bLifterServoPower,
    Enable_Positive := bLifterServoPower,
    Enable_Negative := bLifterServoPower); // Mc_Power

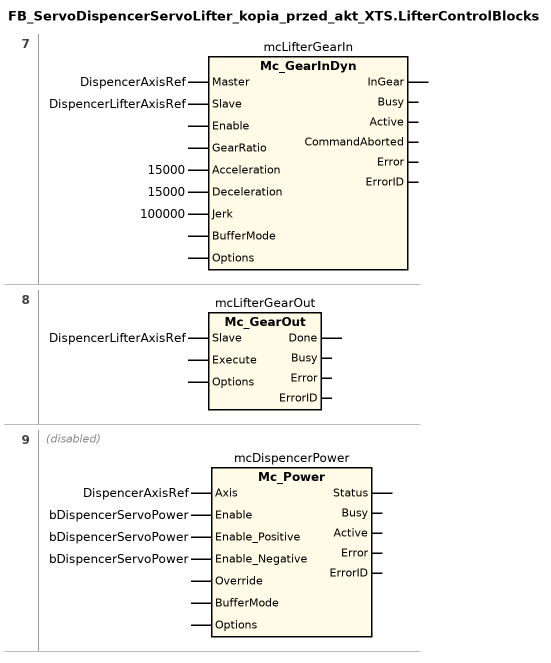
// NETWORK 7
mcLifterGearIn(
    Master := DispencerAxisRef,
    Slave := DispencerLifterAxisRef,
    Acceleration := 15000,
    Deceleration := 15000,
    Jerk := 100000); // Mc_GearInDyn

// NETWORK 8
mcLifterGearOut(Slave := DispencerLifterAxisRef); // Mc_GearOut

// NETWORK 9 (disabled)
// mcDispencerPower(
//     Axis := DispencerAxisRef,
//     Enable := bDispencerServoPower,
//     Enable_Positive := bDispencerServoPower,
//     Enable_Negative := bDispencerServoPower); // Mc_Power
END_ACTION

ACTION Limits:


(*Prędkość dozowania*)
IF mcDispencerMoveAbsolute1.Velocity	 > lrLifterVelocity	THEN		mcDispencerMoveAbsolute1.Velocity	:= lrLifterVelocity;				END_IF
IF mcDispencerMoveAbsolute2.Velocity	 > lrLifterVelocity	THEN		mcDispencerMoveAbsolute2.Velocity	:= lrLifterVelocity;				END_IF

(*Inny parametr*)
//...
END_ACTION

ACTION ManualMovements:
//W trybie ruchów manualnych wykonuj ruchy za pomocą rozkazów manualnych
IF NOT bRun AND NOT (eRunningState=E_DispencerState.ePulling) 
			AND NOT (eRunningState=E_DispencerState.eCleaning) 
THEN
	mcDispencerPower.Override			:=	lrManualOverride;
	mcDispencerManualMove.JogForward	:=	bManualPistonForward;
	mcDispencerManualMove.JogBackwards	:=	bManualPistonBack;
	bSuckingValveActuator				:=	bManualSuckingValve;
	bDosingValveActuator				:=	bManualDosingValve;
	bDropCatcherActuator				:=	bManualDropCatcherForward;
	mcLifterManualMove.JogForward		:=	bManualLifterUp;
	mcLifterManualMove.JogBackwards		:=	bManualLifterDown;
	IF bManualPullingFast OR bManualPullingSlow OR bManualPullingLatch THEN
		bManualPullingLatch				:=	TRUE;
		bDropCatcherActuator			:=	FALSE;
		eRunningState					:=	E_DispencerState.ePulling;
		bManualPullingLatch				:=	FALSE;			
	END_IF	
ELSE	//Kasuje zeby po cyklu nic sie nie poruszało
	IF NOT (eRunningState=E_DispencerState.ePulling) THEN
		mcDispencerMoveAbsolute1.Execute	:=	FALSE;
	END_IF
	mcDispencerManualMove.JogForward		:=	FALSE;
	mcDispencerManualMove.JogBackwards		:=	FALSE;
END_IF


IF bHoming OR bHeightSet THEN
	eState:=E_Station.eHoming;
END_IF
	
Running();

IF NOT bRun THEN
	bCycleDone 					:= FALSE;
	bCycleNotDone 				:= FALSE;	
END_IF
	
ManualMovementsCleaning();
ManualMovementsPulling();

//ZABEZPIECZENIE PRZED UDERZENIEM W TACKĘ OCIEKOWĄ
IF DispencerLifterAxisRef.NcToPlc.ActPos	<	(lrDropCatcherHeightCV+lrDropCatcherOpenDistance) AND NOT bDropCatcherBackSensor THEN
	mcLifterManualMove.JogBackwards:=FALSE;
END_IF

IF (DispencerLifterAxisRef.NcToPlc.ActPos  <= 	lrDropCatcherHeightCV+(lrDropCatcherOpenDistance+5)) (*OR bMultiMasterSyncIn*) THEN //Zmiana XTS
	bDropCatcherActuator:=FALSE;
END_IF
END_ACTION

ACTION ManualMovementsCleaning:

(*****************CYKL MYCIA DOZOWNIKA*******************
eCleaningPreparing:=18,	//Mycie | przejazd do pozycji górnej
eCleaningReady:=19,		//Mycie | pozycja tłoka w górze
eCleaning:=20,			//Mycie | w trakcie ruchu w dół
eCleaningDone:=21		//Mycie | pozycja tłoka w dole
*********************************************************)

// Włączenie mycia
IF bManualCleaningMode  AND  (	NOT (eRunningState	=	E_DispencerState.eCleaningPreparing)		AND
								NOT (eRunningState	=	E_DispencerState.eCleaningReady) 			AND
								NOT (eRunningState	=	E_DispencerState.eCleaning)					AND
								NOT (eRunningState	=	E_DispencerState.eCleaningDone) )			THEN 
	eRunningState	:=	E_DispencerState.eCleaningPreparing;	
END_IF

//Wyłączenie mycia, zatrzymywanie
IF NOT bManualCleaningMode AND  (	eRunningState	=	E_DispencerState.eCleaningReady OR
									eRunningState	=	E_DispencerState.eCleaning OR
									eRunningState	=	E_DispencerState.eCleaningDone )	THEN

	mcDispencerStop.Execute					:= TRUE;
	bSuckingValveActuator					:= FALSE;	
	bDosingValveActuator					:= FALSE;	
	IF 	mcDispencerStop.Done THEN			
		mcDispencerStop.Execute				:= FALSE;
		eState								:= E_Station.eManualMovement;
		eRunningState						:= E_DispencerState.eReady;
	END_IF	
END_IF


//Przygotowanie
IF eRunningState=E_DispencerState.eCleaningPreparing THEN
	bSuckingValveActuator					:= TRUE;
	bDosingValveActuator					:= FALSE;
	mcDispencerMoveAbsolute1.Velocity		:= (lrDosePhase2Velocity*2)		*1.8; 	//Prędkość brana z receptury zwiększona o 30% i 2x większa niż dozowania
	mcDispencerMoveAbsolute1.Acceleration	:= lrDosePhase2Acceleration		*1.8;
	mcDispencerMoveAbsolute1.Deceleration	:= lrDosePhase2Acceleration		*1.8;
	mcDispencerMoveAbsolute1.Position		:= lrRatedDose;
	mcDispencerMoveAbsolute1.Execute		:= bSuckingValveActuator AND bSuckingValveOpenedSensor AND bDosingValveClosedSensor ;
	IF mcDispencerMoveAbsolute1.Done THEN
		mcDispencerMoveAbsolute1.Execute	:= FALSE;
		eRunningState								:= E_DispencerState.eCleaningReady;
	END_IF
END_IF


//Gotowość do mycia
IF eRunningState=E_DispencerState.eCleaningReady THEN
	bSuckingValveActuator					:= FALSE;
	bDosingValveActuator					:= FALSE;
	IF bManualCleaning THEN
		eRunningState								:= E_DispencerState.eCleaning;
	END_IF
END_IF


//Mycie, ruch w dół
IF eRunningState=E_DispencerState.eCleaning THEN
	bSuckingValveActuator					:= FALSE;
	bDosingValveActuator					:= TRUE;
	mcDispencerMoveAbsolute2.Velocity		:= lrDosePhase2Velocity			*1.8;
	mcDispencerMoveAbsolute2.Acceleration	:= lrDosePhase2Acceleration		*1.8;
	mcDispencerMoveAbsolute2.Deceleration	:= lrDosePhase2Acceleration		*1.8;
	mcDispencerMoveAbsolute2.Position		:= 0;
	mcDispencerMoveAbsolute2.Execute		:= bDosingValveActuator AND bSuckingValveClosedSensor AND bDosingValveOpenedSensor;
	IF mcDispencerMoveAbsolute2.Done THEN
		mcDispencerMoveAbsolute2.Execute	:= FALSE;
		eRunningState								:= E_DispencerState.eCleaningDone;
	END_IF	
END_IF


//Koniec mycia
IF eRunningState=E_DispencerState.eCleaningDone THEN
	bSuckingValveActuator					:= FALSE;
	bDosingValveActuator					:= FALSE;
	IF NOT bManualCleaning THEN
		eRunningState								:= E_DispencerState.eCleaningPreparing;
	END_IF
END_IF
END_ACTION

ACTION ManualMovementsPulling:
//CYKL PRZECIĄGANIA MASY
IF eRunningState=E_DispencerState.ePulling THEN
	
	IF NOT bManualPullingFast AND NOT bManualPullingSlow AND NOT bSuckingValveActuator AND NOT bDosingValveActuator AND bSuckingValveClosedSensor AND bDosingValveClosedSensor AND mcDispencerStop.Done THEN
		mcDispencerStop.Execute:=FALSE;
		mcDispencerMoveAbsolute1.Execute:=FALSE;
		mcDispencerMoveAbsolute2.Execute:=FALSE;
		bSuckingValveActuator:=FALSE;
		bDosingValveActuator:=FALSE;
		bManualPullingLatch:=FALSE;
		mcLifterManualMove.JogForward:=FALSE;
		mcLifterManualMove.JogBackwards:= FALSE;
		eState:=E_Station.eManualMovement;
		eRunningState:=E_DispencerState.eReady;
	END_IF

	mcDispencerMoveAbsolute1.Execute:=bSuckingValveActuator AND bSuckingValveOpenedSensor AND bDosingValveClosedSensor AND (bManualPullingFast OR bManualPullingSlow);
	IF mcDispencerMoveAbsolute1.Execute THEN
		;
	END_IF
	mcDispencerMoveAbsolute2.Execute:=bDosingValveActuator AND bSuckingValveClosedSensor AND bDosingValveOpenedSensor AND (bManualPullingFast OR bManualPullingSlow);
	IF bManualPullingFast THEN
		lrPullingVelocity:=300;
	ELSIF bManualPullingSlow THEN
		lrPullingVelocity:=100;
	END_IF
	mcDispencerMoveAbsolute1.Velocity:=lrPullingVelocity;
	mcDispencerMoveAbsolute2.Velocity:=lrPullingVelocity;
	
	mcDispencerMoveAbsolute1.Acceleration:=800;
	mcDispencerMoveAbsolute2.Acceleration:=800;
	mcDispencerMoveAbsolute1.Deceleration:=800;
	mcDispencerMoveAbsolute2.Deceleration:=800;
	mcDispencerMoveAbsolute1.Position:=lrRatedDose;
	mcDispencerMoveAbsolute2.Position:=0;
	
	bSuckingValveActuator:= NOT mcDispencerMoveAbsolute1.DONE AND NOT bDosingValveActuator AND  (bManualPullingFast OR bManualPullingSlow);
	bDosingValveActuator:= NOT mcDispencerMoveAbsolute2.DONE AND NOT bSuckingValveActuator AND (bManualPullingFast OR bManualPullingSlow OR mcDispencerMoveAbsolute2.Busy);
	mcDispencerStop.Execute:=NOT bSuckingValveActuator AND NOT bDosingValveActuator AND NOT bManualPullingFast AND NOT bManualPullingSlow AND eRunningState=E_DispencerState.ePulling;
END_IF
END_ACTION

ACTION Running:
//	100					300			250
IF lrDosePhase1Volume>lrDoseVolume-lrDosePhase2Volume THEN
	lrDosePhase1Volume:=lrDoseVolume-lrDosePhase2Volume;
END_IF
// 200					300			200
IF lrDosePhase2Volume>lrDoseVolume-lrDosePhase1Volume THEN
	lrDosePhase2Volume:=lrDoseVolume-lrDosePhase1Volume;
END_IF


(*Ograniczenia GearRatio*)
lrGearRatio:=-ABS(lrLifterStopDosePosition-lrLifterStartDosePosition+0.000000000001)
							/(*---------------------------------------------------------------------*)
							((BOOL_TO_INT(bLiftSynchroPh1)*lrDosePhase1Volume)
							+(BOOL_TO_INT(bLiftSynchroPh2)*(lrDoseVolume-lrDosePhase2Volume-lrDosePhase1Volume))
							+((BOOL_TO_INT(bLiftSynchroPh3)*lrDosePhase2Volume))
							+ 0.000000000001); 
IF bLiftSynchroPh3 AND lrGearRatio<-1.2THEN
	lrGearRatio:=-1.2;
END_IF
(*Koniec Ograniczenia GearRatio*)

							

CASE eRunningState OF

//====================================
	
	(*Oczekiwanie na wykonanie pojedynczego cyklu*)
	E_DispencerState.eReady:
                                         	
		IF NOT bCycleDone AND NOT bCycleNotDone THEN                                           	
			IF bRun THEN                				
				eRunningState:= E_DispencerState.ePreparingToDose;
				lrSuckingMassStart:=DispencerAxisRef.NcToPlc.ActPos;
			END_IF
		END_IF
		
		bMultiMasterSyncOut:=FALSE;
		
//====================================		
				
	E_DispencerState.ePreparingToDose:

				//Jeśli oś w stanie 'master' przy gearing przejdź do stanu fazy pierwszej dozowania
				IF bDispencerWithLifter THEN
					bDropCatcherActuator:=FALSE;
					mcLifterStop.Execute:=FALSE;
					mcLifterMoveAbsolute.Execute:= NOT mcLifterStop.Done AND bDropCatcherBackSensor AND bDropCatcherActuator=FALSE;
					mcLifterMoveAbsolute.Deceleration:=15000;
					mcLifterMoveAbsolute.Acceleration:=15000;
					mcLifterMoveAbsolute.Velocity:=1100;
					mcLifterMoveAbsolute.Position:=lrLifterStartDosePosition;
				END_IF
				
				mcDispencerStop.Execute:=FALSE;
				//IF ABS(LREAL_TO_DINT(DispencerAxisRef.NcToPlc.ActPos)-LREAL_TO_DINT(lrDoseVolume))>1 THEN //Zmiana dp
					mcDispencerMoveAbsolute1.Execute:= NOT mcDispencerStop.BUSY;
					mcDispencerMoveAbsolute1.Velocity:= lrSuckVelocity;
					mcDispencerMoveAbsolute1.Position:= lrDoseVolume;
					mcDispencerMoveAbsolute1.Acceleration:= lrSuckAcceleration;
					mcDispencerMoveAbsolute1.Deceleration:= lrSuckDeceleration;
				//END_IF;	
				(*n*)
				bMultiMasterSyncOut:=mcDispencerMoveAbsolute1.Done AND ((ABS(DispencerLifterAxisRef.NcToPlc.ActPos)-lrLifterStartDosePosition)<=1);

					//Jeśli osiągnięta pozycja zassania i jeśli jest podnośnik dozownika
					IF (mcLifterMoveAbsolute.Done OR NOT bDispencerWithLifter)  AND (mcDispencerMoveAbsolute1.Done OR ABS(LREAL_TO_DINT(DispencerAxisRef.NcToPlc.ActPos)-LREAL_TO_DINT(lrDoseVolume))<=1(*(LREAL_TO_DINT(DispencerAxisRef.NcToPlc.ActPos)=LREAL_TO_DINT(lrDoseVolume))*)) 
				(*n*)	AND bMultiMasterSyncIn
						THEN
			    	
					//Jeśli nalewarka ma podnośnik i wybrana któraś z opcji ruchu synchronicznego przejdź do procedury zasprzęglania
						IF bDispencerWithLifter AND (bLiftSynchroPh1 OR bLiftSynchroPh2 OR bLiftSynchroPh3) THEN
							mcLifterGearIn.Acceleration:=lrLifterAcceleration;
							mcLifterGearIn.Deceleration:=lrLifterDeceleration;
							mcLifterGearIn.Jerk:=lrLifterDeceleration;
							mcLifterGearIn.GearRatio:=0.0000000001;
						END_IF
						eRunningState:=E_DispencerState.eDosingPh1;
						mcLifterMoveAbsolute.Execute:=FALSE;
						mcDispencerMoveAbsolute1.Execute:= FALSE;
						mcDispencerMoveAbsolute2.Execute:= FALSE;
						mcDispencerMoveAbsolute3.Execute:= FALSE;
						lrStartDosingPos:=DispencerAxisRef.NcToPlc.ActPos;
					END_IF
	
//====================================					
	
	E_DispencerState.eDosingPh1:
				bDropCatcherActuator:=FALSE;
	
				IF bDispencerWithLifter AND (bLiftSynchroPh1 OR bLiftSynchroPh2 OR bLiftSynchroPh3) AND NOT mcLifterGearIn.Enable THEN
					mcLifterGearIn.Enable:= NOT mcDispencerMoveAbsolute1.Busy;
				END_IF
				
				IF (mcLifterGearIn.InGear OR NOT bDispencerWithLifter OR NOT( bLiftSynchroPh1 OR bLiftSynchroPh2 OR bLiftSynchroPh3 )) THEN
					
					mcDispencerMoveAbsolute1.Execute:= bDropCatcherBackSensor;
					mcDispencerMoveAbsolute1.Velocity:= lrDosePhase1Velocity;
					mcDispencerMoveAbsolute1.Position:= lrDoseVolume-lrDosePhase1Volume;
					mcDispencerMoveAbsolute1.Acceleration:= lrDosePhase1Acceleration;
					mcDispencerMoveAbsolute1.Deceleration:= lrDosePhase1Deceleration;
					mcDispencerMoveAbsolute1.BufferMode:= MC_BlendingPrevious;
				END_IF;	
				
				IF bDispencerWithLifter THEN
					IF NOT bLiftSynchroPh1 THEN
						mcLifterGearIn.GearRatio:=0.00000000001;
					ELSE
						mcLifterGearIn.GearRatio:=lrGearRatio;
					END_IF
				END_IF
				//Jeśli zakręcarka na wysokości zakręcania przejdź do stanu zakręcania
				IF (mcLifterGearIn.InGear OR NOT bDispencerWithLifter OR NOT( bLiftSynchroPh1 OR bLiftSynchroPh2 OR bLiftSynchroPh3 )) 
				AND mcDispencerMoveAbsolute1.Execute AND (mcDispencerMoveAbsolute1.Busy OR mcDispencerMoveAbsolute1.Done)
				(*AND lrDosePhase2Volume>lrDosePhase2Volume*) THEN
					
					mcDispencerMoveAbsolute2.Execute:= bDropCatcherBackSensor;
					mcDispencerMoveAbsolute2.Velocity:= lrDosePhase2Velocity;
					mcDispencerMoveAbsolute2.Position:= lrDosePhase2Volume;
					mcDispencerMoveAbsolute2.Acceleration:= lrDosePhase2Acceleration;
					mcDispencerMoveAbsolute2.Deceleration:= lrDosePhase2Deceleration;
					mcDispencerMoveAbsolute2.BufferMode:= MC_BlendingPrevious;
				END_IF
				
				IF mcDispencerMoveAbsolute1.Done AND mcDispencerMoveAbsolute1.Execute THEN
					//mcDispencerMoveAbsolute1.Execute:= FALSE;
					eRunningState:=E_DispencerState.eDosingPh2;
				END_IF
			
	//====================================					
	
	E_DispencerState.eDosingPh2:
	
				IF (mcLifterGearIn.InGear OR NOT bDispencerWithLifter OR NOT( bLiftSynchroPh1 OR bLiftSynchroPh2 OR bLiftSynchroPh3 )) 
					AND mcDispencerMoveAbsolute2.Execute AND (mcDispencerMoveAbsolute2.Busy OR mcDispencerMoveAbsolute2.Done)
							(*AND lrDoseVolume>lrDosePhase2Volume*) THEN	
(*					mcDispencerMoveAbsolute1.Execute:= bDropCatcherBackSensor;
					mcDispencerMoveAbsolute1.Velocity:= lrDosePhase3Velocity;
					mcDispencerMoveAbsolute1.Position:= 0;
					mcDispencerMoveAbsolute1.Acceleration:= lrDosePhase3Acceleration;
					mcDispencerMoveAbsolute1.Deceleration:= lrDosePhase3Deceleration;
					mcDispencerMoveAbsolute1.BufferMode:= MC_BlendingNext;*)
					mcDispencerMoveAbsolute3.Execute:= bDropCatcherBackSensor;
					mcDispencerMoveAbsolute3.Velocity:= lrDosePhase3Velocity;
					mcDispencerMoveAbsolute3.Position:= 0;
					mcDispencerMoveAbsolute3.Acceleration:= lrDosePhase3Acceleration;
					mcDispencerMoveAbsolute3.Deceleration:= lrDosePhase3Deceleration;
					mcDispencerMoveAbsolute3.BufferMode:= MC_BlendingPrevious;
				END_IF
				
				IF bDispencerWithLifter THEN
					IF NOT bLiftSynchroPh2 THEN
						mcLifterGearIn.GearRatio:=0.00000000001;
					ELSE
						mcLifterGearIn.GearRatio:=lrGearRatio;
					END_IF
				END_IF
				
				//IF mcDispencerMoveAbsolute2.Done AND bTest THEN
				IF mcDispencerMoveAbsolute2.Done AND mcDispencerMoveAbsolute2.Execute  THEN					
					//mcDispencerMoveAbsolute2.Execute:= FALSE;
					eRunningState:=E_DispencerState.eDosingPh3;
				END_IF
					
	//====================================	
				
	//FAZA TRZECIA DOZOWANIA
	E_DispencerState.eDosingPh3:
														
		IF bDispencerWithLifter THEN
			IF NOT bLiftSynchroPh3 THEN
				mcLifterGearIn.GearRatio:=0.00000000001;
			ELSE
				mcLifterGearIn.GearRatio:=lrGearRatio;
			END_IF
		END_IF
		(*n*)
		bMultiMasterSyncOut:=NOT mcDispencerMoveAbsolute3.Done;
		
		IF mcDispencerMoveAbsolute3.Done AND (tonDoseValveCloseTimeDec.Q OR bDoseSucking) AND NOT bMultiMasterSyncIn THEN
			
			nCountTest12:=nCountTest12+1;
			lrSuckingMassStart:=DispencerAxisRef.NcToPlc.ActPos;
			mcDispencerMoveAbsolute1.Execute:= FALSE;
			mcDispencerMoveAbsolute2.Execute:= FALSE;
			mcDispencerMoveAbsolute3.Execute:= FALSE;
			IF bDispencerWithLifter THEN (*n*)
				mcLifterGearOut.Execute:=TRUE;
				mcLifterGearIn.Enable:=FALSE;
			END_IF
			IF bDoseSucking THEN (*n*)
				eRunningState:=E_DispencerState.eDoseSucking;
			ELSE
				eRunningState:=E_DispencerState.eGoingUp; 
			END_IF
			
			bDosingValveActuator:=FALSE;
		END_IF
	//====================================	
			
	E_DispencerState.eDoseSucking:
					mcDispencerMoveAbsolute1.Execute:= bDosingValveOpenedSensor AND tonDoseSuckingTimeDelay.Q; // [6] [Podsysanie] Opóźnienie podsysania [ms]
					mcDispencerMoveAbsolute1.Velocity:= 1100;
					mcDispencerMoveAbsolute1.Position:= lrDoseSuckingVolume;
					mcDispencerMoveAbsolute1.Acceleration:= 15000;
					mcDispencerMoveAbsolute1.Deceleration:= 15000;
					IF  mcDispencerMoveAbsolute1.Done THEN
						mcDispencerMoveAbsolute2.Execute:= FALSE;
						mcDispencerMoveAbsolute3.Execute:= FALSE;
					END_IF				
					
					IF bDispencerWithLifter AND tonDoseValveCloseTimeDec.Q THEN	// [2] Opóźnienie zamknięcia zaworu tłoczenia [ms]

						mcLifterMoveAbsolute.Execute:= TRUE; 
						mcLifterMoveAbsolute.Velocity:= 1100;
						mcLifterMoveAbsolute.Position:= lrLifterReadyPosition;
						mcLifterMoveAbsolute.Acceleration:= 15000;
						mcLifterMoveAbsolute.Deceleration:= 15000;

					END_IF
					//DP CZY TUTAJ DODAĆ LIFTER DONE?
					IF mcDispencerMoveAbsolute1.Done AND tonDoseValveCloseTimeDec.Q THEN // [2] Opóźnienie zamknięcia zaworu tłoczenia [ms]		
						eRunningState:=E_DispencerState.eDoseSuckingDone;
						mcDispencerMoveAbsolute1.Execute:= FALSE;
					END_IF		
	

	//====================================

	E_DispencerState.eDoseSuckingDone:
				eRunningState:=E_DispencerState.eGoingUp;
						
		
//====================================					
	
	//DOZOWANIE WYKONANE
	//Zaczyna sie zasysanie i podnoszenie jesli bDispencerWithLifter. Po zaniku bDose, przechodzi do nastepnych stanów	
	E_DispencerState.eGoingUp:
				IF mcLifterGearOut.Done THEN //DP NOWE
					mcLifterGearOut.Execute:=FALSE;
				END_IF
	
				btestgoingup:=btestgoingup+1;
				IF bDispencerWithLifter AND NOT mcLifterGearOut.Done THEN
					IF NOT mcLifterGearInEnable AND NOT mcDispencerMoveAbsolute1.Execute THEN
						mcDispencerMoveAbsolute1.Execute:= bDosingValveClosedSensor AND tonSuckValveOpenTimeDelay.Q; // [3] Opóżnienie rozpoczęcia ssania po tłoczeniu [ms]
						mcDispencerMoveAbsolute1.Velocity:= lrSuckVelocity;
						mcDispencerMoveAbsolute1.Position:= lrDoseVolume;
						mcDispencerMoveAbsolute1.Acceleration:= lrSuckAcceleration;
						mcDispencerMoveAbsolute1.Deceleration:= lrSuckDeceleration;
					END_IF
					mcLifterMoveAbsolute.Execute:= TRUE;
					mcLifterMoveAbsolute.Acceleration:=15000;
					mcLifterMoveAbsolute.Deceleration:=15000;					
					mcLifterMoveAbsolute.Velocity:=1116;
					mcLifterMoveAbsolute.Position:=lrLifterReadyPosition;
					//Koniec ruchu
				ELSE
					mcDispencerMoveAbsolute1.Execute:= bDosingValveClosedSensor;
					mcDispencerMoveAbsolute1.Velocity:= lrSuckVelocity;
					mcDispencerMoveAbsolute1.Position:= lrDoseVolume;
					mcDispencerMoveAbsolute1.Acceleration:= lrSuckAcceleration;
					mcDispencerMoveAbsolute1.Deceleration:= lrSuckDeceleration;
				END_IF
				// [3] Opóżnienie rozpoczęcia ssania po tłoczeniu [ms]
				IF tonSuckValveOpenTimeDelay.Q AND (mcLifterMoveAbsolute.Done OR NOT bDispencerWithLifter) AND (lrLifterActualPosition>lrLifterReadyPosition-5 AND lrLifterActualPosition<lrLifterReadyPosition+5) THEN
						mcLifterMoveAbsolute.Execute:= FALSE;
						eRunningState:=E_DispencerState.eDosingDone;	
				END_IF
  	
//====================================				
		
	E_DispencerState.eDosingDone:
		mcDispencerMoveAbsolute1.Execute:= bDosingValveClosedSensor;
		mcDispencerMoveAbsolute1.Velocity:= lrSuckVelocity;
		mcDispencerMoveAbsolute1.Position:= lrDoseVolume;
		mcDispencerMoveAbsolute1.Acceleration:= lrSuckAcceleration;
		mcDispencerMoveAbsolute1.Deceleration:= lrSuckDeceleration;
		mcDispencerMoveAbsolute1.BufferMode:= MC_Buffered; //ZMIANA BUFFERMODE
			
		IF mcDispencerMoveAbsolute1.Done AND tonSuckValveCloseTimeDelay.Q AND tonDosingDoneDelay.Q THEN // [4] Opóżnienie zamknięcia zaworu ssącego [ms]
			bSuckingValveActuator:=FALSE;
			mcDispencerMoveAbsolute1.Execute:=FALSE;
			eRunningState:=E_DispencerState.eReady;
			bCycleDone := TRUE;
		ELSE
			eRunningState:=E_DispencerState.eSucking;	
		END_IF	
		


//====================================		
	
	E_DispencerState.eSucking:
			mcDispencerMoveAbsolute1.Execute:= bDosingValveClosedSensor; 
			mcDispencerMoveAbsolute1.Velocity:= lrSuckVelocity;
			mcDispencerMoveAbsolute1.Position:= lrDoseVolume;
			mcDispencerMoveAbsolute1.Acceleration:= lrSuckAcceleration;
			mcDispencerMoveAbsolute1.Deceleration:= lrSuckDeceleration;
			IF  mcDispencerMoveAbsolute1.Done AND tonSuckValveCloseTimeDelay.Q AND tonDosingDoneDelay.Q THEN  // [4] Opóżnienie zamknięcia zaworu ssącego [ms]                            
					mcDispencerMoveAbsolute1.Execute:= FALSE;
					mcDispencerMoveAbsolute2.Execute:= FALSE;
					mcDispencerMoveAbsolute3.Execute:= FALSE;
					bSuckingValveActuator:=FALSE;
					mcDispencerMoveAbsolute1.Execute:= FALSE;
					eRunningState:=E_DispencerState.eReady;	
					bCycleDone := TRUE;
			END_IF		

END_CASE
		



		//Tłoczący
		IF eRunningState=E_DispencerState.eDosingPh1 OR eRunningState=E_DispencerState.eDosingPh2 OR eRunningState=E_DispencerState.eDosingPh3 OR 
		   eRunningState=E_DispencerState.eDoseSucking THEN
			
			bDosingValveActuator:= (lrStartDosingPos-lrDosingValveOpenVolume>=LREAL_TO_INT(DispencerAxisRef.NcToPlc.ActPos))AND(lrDosingValveCloseVolume<=LREAL_TO_INT(DispencerAxisRef.NcToPlc.ActPos));
			bSuckingValveActuator:=FALSE;
			
			IF (lrDosingValveOpenVolume+lrDosingValveCloseVolume)>(lrStartDosingPos)  THEN
				bDosingValveActuator:=TRUE;	
				nCheckCount125:=nCheckCount125+1;
			END_IF
			
			IF  lrDoseValveOpenTimeAcc > 0 THEN // [1] Przyśpieszenie otwarcia zaworu tłoczenia [ms]
				bDosingValveActuator:=TRUE;	
				nCheckCount124:=nCheckCount124+1;
			END_IF
										//bylo = (tonDoseValveCloseTimeDec.Q OR bDoseSucking) 
			IF (lrDosingValveCloseVolume>LREAL_TO_INT(DispencerAxisRef.NcToPlc.ActPos)) AND (lrDoseValveCloseTimeDec = 0 AND NOT bDoseSucking) THEN 
				bDosingValveActuator:=FALSE;
				nCheckCount123:=nCheckCount123+1;
			END_IF
			ninttest:=LREAL_TO_INT(DispencerAxisRef.NcToPlc.ActPos);
		END_IF
		
		
		
		//Ssący																								
		IF eRunningState=E_DispencerState.ePreparingToDose OR 
			eRunningState=E_DispencerState.eSucking  OR  
			(*eState=E_DispencerState.eDosingDone OR *)
			eRunningState=E_DispencerState.eGoingUp (*OR
			eState=E_DispencerState.eDoseSuckingDone*) (*AND mcDispencerMoveAbsolute1.Busy*) 
		 THEN
			
			bSuckingValveActuator:=(((ABS(LREAL_TO_INT(lrSuckingMassStart-DispencerAxisRef.NcToPlc.ActPos)))>LREAL_TO_INT(lrSuckValveOpenVolume))
									AND((ABS(LREAL_TO_INT(lrDoseVolume-DispencerAxisRef.NcToPlc.ActPos)))>LREAL_TO_INT(lrSuckValveCloseVolume))); 
																					
			IF lrDoseValveOpenTimeAcc >= 0 THEN // [1] Przyśpieszenie otwarcia zaworu tłoczenia [ms] (Dodatkowe zabezpieczenie bo czasami sie na chwile zamykał)
				bDosingValveActuator:=FALSE;
				nCheckCount1263:=nCheckCount1236+1;
			END_IF 
			
			IF	(lrSuckValveOpenVolume+lrSuckValveCloseVolume)>(ABS(lrDoseVolume-lrSuckingMassStart)) AND (lrSuckValveOpenVolume > mcDispencerMoveAbsolute1.Position) AND 
				(lrSuckValveCloseVolume < mcDispencerMoveAbsolute1.Position)  THEN
				bSuckingValveActuator:=TRUE;	
				nCheckCount1234:=nCheckCount1234+1;
			END_IF
			// [4] Opóżnienie zamknięcia zaworu ssącego [ms]
//dp		IF NOT tonSuckValveCloseTimeDelay.Q AND (eRunningState=E_DispencerState.eDosingDone OR eRunningState=E_DispencerState.eSucking) AND lrSuckValveCloseVolume = 0 THEN (*4*)
			IF NOT tonSuckValveCloseTimeDelay.Q AND (eRunningState=E_DispencerState.eDosingDone OR eRunningState=E_DispencerState.eSucking) AND lrSuckValveCloseVolume = 0 AND (*4*)
			((ABS(LREAL_TO_INT(lrSuckingMassStart-DispencerAxisRef.NcToPlc.ActPos)))>LREAL_TO_INT(lrSuckValveOpenVolume)) THEN
				bSuckingValveActuator:=TRUE;	
				nCheckCount1233:=nCheckCount1233+1;
			END_IF
			//IF NOT tonSuckValveOpenTimeDelay.Q AND eState=E_DispencerState.eGoingUp THEN										
			IF NOT tonSuckValveOpenTimeDelay.Q AND eRunningState=E_DispencerState.eGoingUp THEN
				bSuckingValveActuator:=FALSE;	
				nCountCheckDisp1:=nCountCheckDisp1+1;
			END_IF
			
			IF (lrSuckValveCloseTimeDelay>0 AND tonSuckValveOpenTimeDelay.Q) AND eRunningState=E_DispencerState.eGoingUp THEN
				bSuckingValveActuator:=TRUE;	
				nCheckCount1235:=nCheckCount1235+1;
			END_IF
		END_IF
END_ACTION

ACTION Statistics:

rtrigCycleTimerRead(CLK:=bCycleDone);
IF rtrigCycleTimerRead.Q THEN
		tCycleTime:=tonCycleTimer.ET;
END_IF
tonCycleTimer(IN:=eRunningState>E_DispencerState.eReady,PT:=T#1D);
END_ACTION

END_FUNCTION_BLOCK

// ---- POUs/FB/FileAccess/FB_FileLog.TcPOU
(****************************************************************************************)
(*							Beckhoff Automation Poland									*)
(*								FB_FileLog  v1.0										*)
(*									26.06.2014											*)
(*			Blok funkcyjny pozwalający logowac dane do pliku							*)
(*	Uwaga - blok nie posiada reakcji na zbocze narastajace,								*)
(*	aby mogl byc wykorzystany wielokrotnie w jednym cyklu programu. 					*)
(*	Reakcja na zbocze musi byc wykonana na zewnatrz bloku. 								*)
(*	W przypadku pojawiania sie komunikatow czesciej niz blok jest w stanie zapisac,		*)
(*	dane sa buforowane w pamieci w zmiennej 											*)
 (*	arrSaveEventBuffer:ARRAY [1..20] OF STRING; 										*)
(*______________________________________________________________________________________*)
FUNCTION_BLOCK FB_FileLog
VAR_INPUT
	bAdd					: BOOL;			(* Dodaj wpis *)
	sMessage				: STRING(1000);	(* Tresc wpisu *)
	bNoAndTime				: BOOL:= TRUE; (* TRUE - dodaj nr porzadkowy i stempel czasowy *)
	sActTime				: STRING;		(* Aktualny czas *)
(* Ustawienia zapisu do pliku *)
	AmsNetId				: T_AmsNetId;	(* AMS NET ID obiektu docelowego, gdy lokalnie, to zmienna moze byc pusta *)
	sPath					: STRING; 		(* Sciezka pliku, np  'Hard Disk\'*)
	sName					: STRING; 		(* Nazwa pliku wraz z rozszerzeniem 'LogFile.txt'; *)
END_VAR
VAR_OUTPUT
	bBusy					: BOOL;
	bError					: BOOL;
END_VAR
VAR
(* Logowanie do plików *)
	fbSaveEvent: 			FB_SaveTextToFile;
	fbSaveEventBuffer:		FB_MemRingBuffer;
	arrSaveEventBuffer: 	ARRAY [1..20] OF STRING(1000);
	wMessageNo: 			WORD;
	sFileMessage: 			STRING(1000);
	nStep: 					BYTE;
END_VAR

fbSaveEventBuffer(
	pWrite:= ADR(sMessage),
	cbWrite:= SIZEOF(sMessage),
	pRead:= ADR(sFileMessage),
	cbRead:= SIZEOF(sFileMessage),
	pBuffer:= ADR(arrSaveEventBuffer),
	cbBuffer:= SIZEOF(arrSaveEventBuffer),
	bOk=> ,
	nCount=> , 
	cbSize=> , 
	cbReturn=> );
IF bAdd THEN
	IF bNoAndTime THEN
		wMessageNo:=wMessageNo + 1;
		sMessage := CONCAT(CONCAT(CONCAT(CONCAT(CONCAT(WORD_TO_STRING(wMessageNo),'.$t'),sActTime),'$t'),sMessage),'$n');
	END_IF
	fbSaveEventBuffer.A_AddTail();
END_IF

CASE nStep OF
	0:
	(* Jesli jest komunikat do zapisania to zapisz *)
	IF fbSaveEventBuffer.nCount>0 THEN
		fbSaveEventBuffer.A_RemoveHead();
		fbSaveEvent.bExecute:=TRUE;
		nStep := nStep + 10;
	END_IF
	10:
	fbSaveEvent.bExecute:=FALSE;
	(* Jak zapis zakonczony sukcesem - to wroc do kroku 0 *)
	IF NOT bBusy AND NOT bError THEN
		nStep := 0;
	END_IF
	(* Jak blad to zresetuj bloczek i podejmij próbę ponownie *)
	IF bError THEN
		nStep := nStep + 10;
	END_IF
	20:
		fbSaveEvent.bExecute:=TRUE;
		nStep := nStep - 10;
END_CASE

fbSaveEvent(
	AmsNetId	:= AmsNetId,
	sPath		:= sPath,
	sName		:= sName,
	sLine		:= sFileMessage,
	bBusy		=> bBusy,
	bError		=> bError);

END_FUNCTION_BLOCK

// ---- POUs/FB/NewFBs/FB_SensorAcetone.TcPOU
FUNCTION_BLOCK FB_SensorAcetone
VAR_INPUT
	bEnable										:	BOOL;
	bReset										:	BOOL;
	bWarningAcknowledge							:	BOOL;
	bSensorAcetoneDetectionError			 	:	BOOL;			//Czujnik detekcji acetonu usterka bład
	bSensorAcetoneDetectionLevel2			 	:	BOOL;			// Alarm poziomu 2 detekcja acetonu 40%DGW (dolna granica wybuchowści)
	bSensorAcetoneDetectionLevel1				:	BOOL;			// Alarm poziomu 1 detekcja acetonu 20%DGW (dolna granica wybuchowści)
	iStationIndex								:	UDINT;
END_VAR
VAR_OUTPUT
	bError										:	BOOL;
	bWarning									:	BOOL;
	
	nErrorNr									: 	UDINT;							//Nr błędu grzałki zasadniczej
	sStationName								: 	STRING(200);
	sErrorDescription							: 	STRING(200);	
	sErrorDescription2							: 	STRING(200);	
	udiStationID								:	UDINT;				// Nr stacji		
	sWarningDescription							: 	STRING(200);	

END_VAR
VAR
END_VAR

ACT_Cycle();
aStationID();

ACTION ACT_Cycle:
IF (bReset) THEN
	bError 							:= FALSE;
	sErrorDescription 				:= '';
	sErrorDescription2 				:= '';
	nErrorNr						:= 0;
END_IF

IF bWarningAcknowledge THEN
		bWarning					:= FALSE;
		sWarningDescription			:= '';
END_IF

IF (bEnable) THEN
	IF (bSensorAcetoneDetectionError) THEN
		bError 						:= TRUE;
		sStationName				:= 'Czujnik gazów łatwopalnych';
		sErrorDescription			:= 'Błąd czujnika gazu';
		sErrorDescription2			:= 'Wymagany ręczny reset czujnika';
		nErrorNr					:= 365;
	ELSIF (bSensorAcetoneDetectionLevel2 AND NOT bError) THEN
		bError 						:= TRUE;
		sStationName				:= 'Czujnik gazów łatwopalnych';
		sErrorDescription			:= 'Alarm poziomu 2 detekcja gazu 40%DGW';
		sErrorDescription2			:= 'Blokada czujnika gazów - sprawdź stan i zresetuj ręcznie przyciskiem na czujniku';
		nErrorNr					:= 366;
	END_IF

	IF (bSensorAcetoneDetectionLevel1 AND NOT bWarning) THEN
		bWarning 					:= TRUE;
		sWarningDescription			:= 'Alarm poziomu 1 detekcja gazu 10%DGW';
	END_IF
END_IF
END_ACTION

ACTION aStationID:
udiStationID	:=	iStationIndex;
END_ACTION

END_FUNCTION_BLOCK

// ---- POUs/FB/POUsAxisOnline/AX5000/FB_AxisDiag.TcPOU
//==================================================================================================
//							Beckhoff Automation Poland
//								23.05.2018
//					Blok do diagnostyki osi
// 	v1.1	|| TC v 3.1.4022.16	|| - optymalizacja kodu
// 	v1.0	|| TC v 3.1.4020.0	|| - pierwsza wersja
//==================================================================================================
FUNCTION_BLOCK FB_AxisDiag
VAR_INPUT
	IPCNetID							: T_AmsNetId; 	(* AmsNetId of the IPC *)
	Timeout								: TIME := DEFAULT_ADS_TIMEOUT;
	Reset								: BOOL;
	GetDiag								: BOOL;
END_VAR
VAR_IN_OUT
	Axis	 							: AXIS_REF;
	stAX5000Diag						: ST_AX5000Diag;
END_VAR
VAR_OUTPUT
	Error								: BOOL;
	AdsErrId							: UINT;
	SercosErrId							: UINT;
	ResetAct							: BOOL;
	DiagAct								: BOOL;
	Busy								: BOOL;
END_VAR
VAR
	iState								: INT;
	iSubState							: INT;
	GetDriveRef							: BOOL;
	DriveRef								: ST_DriveRef; (* contains sNetID of EcMaster, nSlaveAddr of EcDrive, nDriveNo of EcDrive, either preset or read from NC *)
	AxisID								: UDINT;

	C1DErrorPrev							: BOOL;
	WcStateErrorPrev						: BOOL;
	AxisErrorPrev							: BOOL;
	OperationalPrev						: BOOL;
	ResetPrev							: BOOL;
	GetDiagPrev							: BOOL;

	fbSoERead							: FB_SoERead;
	fbDiagMessage 						: FB_SoEReadDiagMessage;
	fbClassXDiag							: FB_SoEReadClassXDiag;
	fbDiagNumber						: FB_SoEReadDiagNumber;
	fbDiagNumberList						: FB_SoEReadDiagNumberList;

	fbReset								: FB_SoEReset;
	fbDelay								: TON;
	fbGetSlaveState 						: FB_EcGetSlaveState;
	fbReqSlaveState 						: FB_EcReqSlaveState;
	fbNcReset 							: MC_Reset;

	fbAdsRead							: ADSREAD;
	readBuffer							: ARRAY[0..9] OF BYTE;
	Ids									: T_AmsNetIdArr;
	strSoEString							: ST_SoE_String;
END_VAR
VAR CONSTANT
	NCIDXG_AXPARMS					: UDINT := 16#00004000;	(* Axis with ID: Parameter 			*)
	NCIDXO_AXP_HWAMSADDR			: UDINT := 16#00000031;
END_VAR

stAX5000Diag.bOperational	:= Axis.NcToPlc.StateDWord.0;
stAX5000Diag.bC1DError	 	:= Axis.NcToPlc.StateDWord.28;
stAX5000Diag.bWcStateError 	:= Axis.NcToPlc.StateDWord.30;
stAX5000Diag.bAxisError		:= Axis.NcToPlc.StateDWord.31;
stAX5000Diag.iAxisErrorCode	:= Axis.NcToPlc.ErrorCode;

CASE iState OF
0:	(* idle *)
	GetDriveRef 	:= (DriveRef.nSlaveAddr = 0);

	IF GetDriveRef THEN
		Busy			:= TRUE;
		Error			:= FALSE;
		AdsErrId		:= 0;
		SercosErrId		:= 0;
		iState 			:= 1;
		iSubState		:= 0;
		AxisID 			:= Axis.NcToPlc.AxisId;

	ELSIF Reset AND NOT ResetPrev THEN
		Busy			:= TRUE;
		ResetAct		:= TRUE;
		ResetPrev		:= Reset;
		Error			:= FALSE;
		AdsErrId		:= 0;
		SercosErrId		:= 0;
		iState 			:= 2;
		iSubState		:= 0;
		AxisID 			:= Axis.NcToPlc.AxisId;

	ELSIF GetDiag AND NOT GetDiagPrev OR
		(stAX5000Diag.bC1DError AND NOT C1DErrorPrev) OR (NOT stAX5000Diag.bC1DError AND C1DErrorPrev) (* rising/falling C1D *) OR
		(stAX5000Diag.bWcStateError AND NOT WcStateErrorPrev) OR (NOT stAX5000Diag.bWcStateError AND WcStateErrorPrev) (* rising/falling WcState *) OR
		(stAX5000Diag.bAxisError AND NOT AxisErrorPrev) OR (NOT stAX5000Diag.bAxisError AND AxisErrorPrev) (* rising/falling NcError *) OR
		(stAX5000Diag.bOperational AND NOT OperationalPrev) OR (NOT stAX5000Diag.bOperational AND OperationalPrev) (* rising/falling Enable *) THEN

		Busy			:= TRUE;
		DiagAct			:= TRUE;
		GetDiagPrev		:= GetDiag;
		Error			:= FALSE;
		AdsErrId		:= 0;
		SercosErrId		:= 0;
		iState 			:= 3;
		iSubState		:= 0;
		AxisID 			:= Axis.NcToPlc.AxisId;

		(* set/clear flags *)
		C1DErrorPrev		:= stAX5000Diag.bC1DError;
		WcStateErrorPrev	:= stAX5000Diag.bWcStateError;
		AxisErrorPrev		:= stAX5000Diag.bAxisError;
		OperationalPrev		:= stAX5000Diag.bOperational;

	ELSE
		ResetAct	:= FALSE;
		DiagAct		:= FALSE;
	END_IF

1:	(* get drive reference *)
	M_GetDriveRef();

2:	(* reset and state change *)
	M_Reset();

3:	(* get diag data *)
	M_GetDiagnosis();

END_CASE

(* clear latch *)
ResetPrev	:= ResetPrev AND Reset;
GetDiagPrev	:= GetDiagPrev AND GetDiag;

ACTION M_GetDiagnosis:
CASE iSubState OF
0:	fbClassXDiag(
		NetId		:= IPCNetID,
		Execute		:= TRUE,
		DiagClass 	:= 1,
		Timeout		:= DEFAULT_ADS_TIMEOUT,
		Axis		:= Axis,
	);

	IF NOT fbClassXDiag.Busy THEN
		fbClassXDiag(Execute:= FALSE,Axis := Axis);

		IF NOT fbClassXDiag.Error THEN
			stAX5000Diag.wClass1Diag	:= fbClassXDiag.ClassXDiag;
			stAX5000Diag.stClass1Diag	:= F_ConvWordToSTAX5000C1D(stAX5000Diag.wClass1Diag);
		ELSE
			Error			:= TRUE;
			AdsErrId		:= fbClassXDiag.AdsErrId;
			SercosErrId	:= fbClassXDiag.SercosErrId;
		END_IF
		iSubState	:= iSubState + 1;
	END_IF

1:	fbDiagMessage(
		NetId	:= IPCNetID,
		Execute	:= TRUE,
		Timeout	:= DEFAULT_ADS_TIMEOUT,
		Axis	:= Axis,
	);

	IF NOT fbDiagMessage.Busy THEN
		fbDiagMessage(Execute:= FALSE,Axis := Axis);

		IF NOT fbDiagMessage.Error THEN
			stAX5000Diag.strDiagMessage := LEFT(fbDiagMessage.DiagMessage.strData, UINT_TO_INT(fbDiagMessage.DiagMessage.iActualSize));
		ELSE
			Error			:= TRUE;
			AdsErrId		:= fbDiagMessage.AdsErrId;
			SercosErrId	:= fbDiagMessage.SercosErrId;
		END_IF
		iSubState	:= iSubState + 1;
	END_IF

2:	fbDiagNumber(
		NetId	:= IPCNetID,
		Execute	:= TRUE,
		Timeout	:= DEFAULT_ADS_TIMEOUT,
		Axis	:= Axis,
	);

	IF NOT fbDiagNumber.Busy THEN
		fbDiagNumber(Execute:= FALSE,Axis := Axis);

		IF NOT fbDiagNumber.Error THEN
			stAX5000Diag.iDiagNumber := fbDiagNumber.DiagNumber;
		ELSE
			Error			:= TRUE;
			AdsErrId		:= fbDiagNumber.AdsErrId;
			SercosErrId	:= fbDiagNumber.SercosErrId;
		END_IF
		iSubState	:= iSubState + 1;
	END_IF

3:	fbSoERead(
		NetId	:= IPCNetID,
		Execute	:= TRUE,
		Idn		:= 135,
		Element	:=16#44,
		pDstBuf	:=ADR(stAX5000Diag.wDriveStatus),
		BufLen	:=SIZEOF(stAX5000Diag.wDriveStatus),
		Timeout	:= DEFAULT_ADS_TIMEOUT,
		Axis	:= Axis,
	);

	IF NOT fbSoERead.Busy THEN
		fbSoERead(Execute:= FALSE,Axis := Axis);
		IF NOT fbSoERead.Error THEN
			stAX5000Diag.stDriveStatus := F_ConvWordToSTAX5000DriveStatus(stAX5000Diag.wDriveStatus);
			iSubState		:= iSubState + 1;
		ELSE
			Error			:= TRUE;
			AdsErrId		:= fbSoERead.AdsErrId;
			SercosErrId	:= fbSoERead.SercosErrId;
			iSubState		:= iSubState + 2;
		END_IF
	END_IF

4:	fbSoERead(
		NetId	:= IPCNetID,
		Execute	:= TRUE,
		Idn		:= stAX5000Diag.stDriveStatus.iActOpModeParNum,
		Element	:=16#44,
		pDstBuf	:=ADR(stAX5000Diag.stDriveStatus.eActOpMode),
		BufLen	:=SIZEOF(stAX5000Diag.stDriveStatus.eActOpMode),
		Timeout	:= DEFAULT_ADS_TIMEOUT,
		Axis	:= Axis,
	);

	IF NOT fbSoERead.Busy THEN
		fbSoERead(Execute:= FALSE,Axis := Axis);
		IF NOT fbSoERead.Error THEN
			;
		ELSE
			Error			:= TRUE;
			AdsErrId		:= fbSoERead.AdsErrId;
			SercosErrId	:= fbSoERead.SercosErrId;
		END_IF
		iSubState	:= iSubState + 1;
	END_IF

5:	fbGetSlaveState(
		sNetId		:= DriveRef.sNetId,
		nSlaveAddr	:= DriveRef.nSlaveAddr,
		bExecute	:= TRUE,
		tTimeout	:= DEFAULT_ADS_TIMEOUT,
	);

	IF NOT fbGetSlaveState.bBusy THEN
		fbGetSlaveState(bExecute:= FALSE);
		IF NOT fbGetSlaveState.bError THEN
			stAX5000Diag.stEcSlaveState := fbGetSlaveState.state;
			stAX5000Diag.stEcSlaveStateBits := F_ConvSlaveStateToBits(fbGetSlaveState.state);
		ELSE
			Error			:= TRUE;
			AdsErrId		:= UDINT_TO_UINT(fbGetSlaveState.nErrId);
		END_IF

		IF stAX5000Diag.stEcSlaveStateBits.bError THEN
			IF stAX5000Diag.stEcSlaveStateBits.bPreop THEN
				(* read S21 - IDN List of Invalid operation data for CP2 (Preop->SaveOp) *)
				MEMSET(ADR(stAX5000Diag.stCPxInvParamList), 0, SIZEOF(stAX5000Diag.stCPxInvParamList));
				stAX5000Diag.bPreopToSafeOpError := TRUE;
				stAX5000Diag.bSafeOpToOpError := FALSE;
				iSubState	:= iSubState + 1;
			ELSIF stAX5000Diag.stEcSlaveStateBits.bSafeOp THEN
				(* read S22 - IDN List of Invalid operation data for CP3 (SaveOp->Op) *)
				MEMSET(ADR(stAX5000Diag.stCPxInvParamList), 0, SIZEOF(stAX5000Diag.stCPxInvParamList));
				stAX5000Diag.bPreopToSafeOpError := FALSE;
				stAX5000Diag.bSafeOpToOpError := TRUE;
				iSubState	:= iSubState + 2;
			ELSE
				(* Skip S21 + S22 *)
				MEMSET(ADR(stAX5000Diag.stCPxInvParamList), 0, SIZEOF(stAX5000Diag.stCPxInvParamList));
				stAX5000Diag.bPreopToSafeOpError := FALSE;
				stAX5000Diag.bSafeOpToOpError := FALSE;
				iSubState	:= iSubState + 3;
			END_IF
		ELSE
			(* Skip S21 + S22 *)
			MEMSET(ADR(stAX5000Diag.stCPxInvParamList), 0, SIZEOF(stAX5000Diag.stCPxInvParamList));
			stAX5000Diag.bPreopToSafeOpError := FALSE;
			stAX5000Diag.bSafeOpToOpError := FALSE;
			iSubState	:= iSubState + 3;
		END_IF
	END_IF

6:	(* read S21 - IDN List of Invalid operation data for CP2 (Preop->SaveOp) *)
	fbSoERead(
		NetId	:= IPCNetID,
		Execute	:= TRUE,
		Idn		:= 21,
		Element	:=16#40,
		pDstBuf	:=ADR(stAX5000Diag.stCPxInvParamList),
		BufLen	:=SIZEOF(stAX5000Diag.stCPxInvParamList),
		Timeout	:= DEFAULT_ADS_TIMEOUT,
		Axis	:= Axis,
	);

	IF NOT fbSoERead.Busy THEN
		fbSoERead(Execute:= FALSE,Axis := Axis);
		IF NOT fbSoERead.Error THEN
			;
		ELSE
			Error			:= TRUE;
			AdsErrId		:= fbSoERead.AdsErrId;
			SercosErrId	:= fbSoERead.SercosErrId;
		END_IF
		iSubState	:= iSubState + 2;
	END_IF

7:	(* read S22 - IDN List of Invalid operation data for CP3 (SaveOp->Op) *)
	fbSoERead(
		NetId	:= IPCNetID,
		Execute	:= TRUE,
		Idn		:= 22,
		Element	:=16#40,
		pDstBuf	:=ADR(stAX5000Diag.stCPxInvParamList),
		BufLen	:=SIZEOF(stAX5000Diag.stCPxInvParamList),
		Timeout	:= DEFAULT_ADS_TIMEOUT,
		Axis	:= Axis,
	);

	IF NOT fbSoERead.Busy THEN
		fbSoERead(Execute:= FALSE,Axis := Axis);
		IF NOT fbSoERead.Error THEN
			;
		ELSE
			Error			:= TRUE;
			AdsErrId		:= fbSoERead.AdsErrId;
			SercosErrId	:= fbSoERead.SercosErrId;
		END_IF
		iSubState	:= iSubState + 1;
	END_IF

8:	fbDiagNumberList(
		NetId			:= IPCNetID,
		Execute			:= TRUE,
		Timeout			:= DEFAULT_ADS_TIMEOUT,
		pDiagNumber		:= ADR(stAX5000Diag.stDiagNumberList),
		Size			:= SIZEOF(stAX5000Diag.stDiagNumberList),
		Axis			:= Axis,
	);

	IF NOT fbDiagNumberList.Busy THEN
		fbDiagNumberList(Execute:= FALSE,Axis := Axis);

		IF fbDiagNumberList.Error THEN
			Error			:= TRUE;
			AdsErrId		:= fbDiagNumberList.AdsErrId;
			SercosErrId	:= fbDiagNumberList.SercosErrId;
		END_IF

		IF (stAX5000Diag.strMotorType = '') OR (stAX5000Diag.strDriveType = '') THEN
			iSubState	:= iSubState + 1;
		ELSE
			DiagAct	:= FALSE;
			iSubState	:= 0;
			iState		:= 0;
			Busy		:= FALSE;
		END_IF
	END_IF

9:	fbSoERead(
		NetId	:= IPCNetID,
		Execute	:= TRUE,
		Idn		:= P_0_IDN + 53,
		Element	:=16#44,
		pDstBuf	:=ADR(strSoEString),
		BufLen	:=SIZEOF(strSoEString),
		Timeout	:= DEFAULT_ADS_TIMEOUT,
		Axis	:= Axis,
	);

	IF NOT fbSoERead.Busy THEN
		fbSoERead(Execute:= FALSE,Axis := Axis);
		IF NOT fbSoERead.Error THEN
			MEMSET(ADR(stAX5000Diag.strMotorType),0,SIZEOF(stAX5000Diag.strMotorType));
			MEMCPY(ADR(stAX5000Diag.strMotorType),ADR(strSoEString.strData),MIN(SIZEOF(stAX5000Diag.strMotorType),strSoEString.iActualSize));
		ELSE
			Error			:= TRUE;
			AdsErrId		:= fbSoERead.AdsErrId;
			SercosErrId	:= fbSoERead.SercosErrId;
		END_IF
		iSubState	:= iSubState + 1;
	END_IF

10:	fbSoERead(
		NetId	:= IPCNetID,
		Execute	:= TRUE,
		Idn		:= P_0_IDN + 324,
		Element	:=16#44,
		pDstBuf	:=ADR(strSoEString),
		BufLen	:=SIZEOF(strSoEString),
		Timeout	:= DEFAULT_ADS_TIMEOUT,
		Axis	:= Axis,
	);

	IF NOT fbSoERead.Busy THEN
		fbSoERead(Execute:= FALSE,Axis := Axis);
		IF NOT fbSoERead.Error THEN
			MEMSET(ADR(stAX5000Diag.strDriveType),0,SIZEOF(stAX5000Diag.strDriveType));
			MEMCPY(ADR(stAX5000Diag.strDriveType),ADR(strSoEString.strData),MIN(SIZEOF(stAX5000Diag.strDriveType),strSoEString.iActualSize));
		ELSE
			Error			:= TRUE;
			AdsErrId		:= fbSoERead.AdsErrId;
			SercosErrId	:= fbSoERead.SercosErrId;
		END_IF
		DiagAct	:= FALSE;
		iSubState	:= 0;
		iState		:= 0;
		Busy		:= FALSE;
	END_IF


END_CASE
END_ACTION

ACTION M_GetDriveRef:
(* get reference from NC *)
fbAdsRead(
	NETID	:= IPCNetID,
	PORT	:= AMSPORT_R0_NC,
	IDXGRP	:= NCIDXG_AXPARMS + Axis.NcToPlc.AxisId,
	IDXOFFS	:= NCIDXO_AXP_HWAMSADDR,
	LEN		:= SIZEOF(readBuffer) ,
	DESTADDR:= ADR(readBuffer),
	READ	:= TRUE,
	TMOUT	:= Timeout
);

IF NOT fbAdsRead.BUSY THEN
	fbAdsRead(READ := FALSE);
	stAX5000Diag.nNCAxisID := Axis.NcToPlc.AxisId;

	IF NOT fbAdsRead.ERR THEN
		MEMCPY(ADR(Ids), ADR(readBuffer), SIZEOF(Ids)); 										(* readBuffer[0..5] *)
		MEMCPY(ADR(DriveRef.nSlaveAddr), ADR(readBuffer[6]), SIZEOF(DriveRef.nSlaveAddr));  	(* readBuffer[6..7] *)
		MEMCPY(ADR(DriveRef.nDriveNo), ADR(readBuffer[8]), SIZEOF(DriveRef.nDriveNo));  		(* readBuffer[8..9] *)

		(* create string out of byte array *)
		DriveRef.sNetId := F_CreateAmsNetId(Ids);
		GetDriveRef := FALSE;
	END_IF

	Busy	:= FALSE;
	iState	:= 0;
END_IF
END_ACTION

ACTION M_Reset:
CASE iSubState OF
0:
	IF stAX5000Diag.bWcStateError OR stAX5000Diag.bC1DError THEN
		(* ResetAmplifier *)
		iSubState := iSubState + 1;
	ELSIF (NOT stAX5000Diag.bOperational) OR stAX5000Diag.bAxisError OR (stAX5000Diag.iAxisErrorCode <> 0) THEN
		(* NC Reset only *)
		iSubState := 6;
	ELSE
		(* reset not required *)
		iSubState	:= 0;
		iState		:= 0;
		Busy		:= FALSE;
		ResetAct	:= FALSE;
	END_IF

1:	(* ResetAmplifier *)
	fbReset(
		NetId	:= IPCNetID,
		Execute	:= TRUE,
		Timeout	:= DEFAULT_ADS_TIMEOUT,
		Axis	:= Axis,
	);
	IF NOT fbReset.Busy THEN
		fbReset(Execute:= FALSE, Axis:= Axis);

		IF NOT fbReset.Error THEN
			iSubState	:= iSubState + 1;
		ELSE
			Error			:= TRUE;
			AdsErrId		:= fbReset.AdsErrId;
			SercosErrId		:= fbReset.SercosErrId;
			Busy			:= FALSE;
			ResetAct		:= FALSE;
			iSubState		:= 0;
			iState			:= 0;
		END_IF
	END_IF

2:	fbDelay(IN:=TRUE, PT:=t#3s);
	IF fbDelay.Q THEN
		fbDelay(IN:=FALSE);
		iSubState	:= iSubState + 1;
	END_IF

3:	fbGetSlaveState(
		sNetId		:= DriveRef.sNetId,
		nSlaveAddr	:= DriveRef.nSlaveAddr,
		bExecute	:= TRUE,
		tTimeout	:= DEFAULT_ADS_TIMEOUT,
	);

	IF NOT fbGetSlaveState.bBusy THEN
		fbGetSlaveState(bExecute:= FALSE);

		IF NOT fbGetSlaveState.bError THEN
			IF Axis.NcToPlc.StateDWord.31 OR (Axis.NcToPlc.ErrorCode <> 0) THEN
				iSubState	:= 6;
			ELSE
				Busy		:= FALSE;
				ResetAct	:= FALSE;
				iSubState	:= 0;
				iState		:= 0;
			END_IF
		ELSE
			Error			:= TRUE;
			AdsErrId		:= UDINT_TO_UINT(fbGetSlaveState.nErrId);
			Busy			:= FALSE;
			ResetAct		:= FALSE;
			iSubState		:= 0;
			iState			:= 0;
		END_IF
	END_IF

5:	(* set op *)
	fbReqSlaveState(
		sNetId		:= DriveRef.sNetId,
		nSlaveAddr	:= DriveRef.nSlaveAddr,
		bExecute	:= TRUE,
		tTimeout	:= DEFAULT_ADS_TIMEOUT,
		state		:= EC_DEVICE_STATE_OP);

	IF NOT fbReqSlaveState.bBusy THEN
		fbReqSlaveState(bExecute:= FALSE);

		IF NOT fbReqSlaveState.bError THEN
			iSubState	:= iSubState + 1;
		ELSE
			Error		:= TRUE;
			AdsErrId	:= UDINT_TO_UINT(fbReqSlaveState.nErrId);
			Busy		:= FALSE;
			ResetAct	:= FALSE;
			iSubState	:= 0;
			iState		:= 0;
		END_IF
	END_IF

6:	fbNcReset(
		Execute:= TRUE,
		Axis:= Axis,
	);
	IF fbNcReset.Done OR fbNcReset.Error THEN
		IF fbNcReset.Error THEN
			Error 		:= TRUE;
			AdsErrId 	:= UDINT_TO_UINT(fbNcReset.ErrorID);
		END_IF

		iSubState	:= 0;
		iState		:= 0;
		Busy		:= FALSE;
		ResetAct	:= FALSE;
		fbNcReset(Execute:= FALSE, Axis:= Axis);
	END_IF
END_CASE
END_ACTION

END_FUNCTION_BLOCK

// ---- POUs/FB/POUsAxisOnline/AX5000/FB_ChangeEtherCATSlaveState.TcPOU
//==================================================================================================
//							Beckhoff Automation Poland
//									23.05.2018
//	Blok zmienia stan EtherCAT Slave i monitoruje flage ukonczenia
//
//	Niezbedne biblioteki: Tc2_EtherCAT
//
// 	v1.1	|| TC v 3.1.4022.16	|| - optymalizacja kodu
// 	v1.0	|| TC v 3.1.4020.32	|| - pierwsza wersja
//==================================================================================================
FUNCTION_BLOCK FB_ChangeEtherCATSlaveState
VAR_INPUT
	bExecute								: BOOL;							// Start on rising edge
	sEtherCAT_NetID							: STRING;						// EtherCAT Master NetID
	nSlaveAddr								: UINT;							// EtherCAT Drive slave port
	byReguestedState						: BYTE;							(* 	16#1- EC_DEVICE_STATE_INIT  
																				16#2- EC_DEVICE_STATE_PREOP     
																				16#3- EC_DEVICE_STATE_BOOTSTRAP     
																				16#4- EC_DEVICE_STATE_SAFEOP  
																				16#8- EC_DEVICE_STATE_OP
																				16#10- EC_DEVICE_STATE_ERROR  *)
END_VAR
VAR_OUTPUT
	byActualState							: BYTE;							(* 	16#1-EC_DEVICE_STATE_INIT  
																				16#2-EC_DEVICE_STATE_PREOP     
																				16#3-EC_DEVICE_STATE_BOOTSTRAP     
																				16#4-EC_DEVICE_STATE_SAFEOP  
																				16#8-EC_DEVICE_STATE_OP
																				16#10-EC_DEVICE_STATE_ERROR  *)
	bBusy									: BOOL;
	bDone									: BOOL;
	bError									: BOOL;
	udiErrorID								: UDINT;	
END_VAR
VAR	
	fbEcReqSlaveState						: FB_EcReqSlaveState;
	fbEcGetSlaveState						: FB_EcGetSlaveState;
	timerTON								: TON;
	rtExecute								: R_TRIG;
	iState									: INT;
	iTry									: INT;							// number of tries
END_VAR

timerTON(PT:=T#500MS);
rtExecute(CLK:=bExecute);

CASE iState OF

	0:																// Init parameters
		IF rtExecute.Q THEN
			bBusy							:= TRUE;
			bDone							:= FALSE;
			bError							:= FALSE;
			udiErrorID						:= 0;
			iTry							:= 0;
			fbEcReqSlaveState.sNetId		:= sEtherCAT_NetID; 
			fbEcGetSlaveState.sNetId		:= sEtherCAT_NetID; 
			fbEcReqSlaveState.nSlaveAddr	:= nSlaveAddr; 
			fbEcGetSlaveState.nSlaveAddr	:= nSlaveAddr;
			fbEcReqSlaveState.state			:= byReguestedState;
			fbEcReqSlaveState.bExecute		:= TRUE;
			iState							:= iState + 10;			
		END_IF
		
	10:																// State request
		fbEcReqSlaveState.bExecute			:= FALSE;
		IF NOT fbEcReqSlaveState.bBusy THEN
			IF fbEcReqSlaveState.bError THEN
				iState						:= 99;
			ELSE
				iState						:= iState + 10;
			END_IF
		END_IF

		
	20:																// Request every 0.5s
		timerTON.IN							:= TRUE;
		IF timerTON.Q THEN
			timerTON.IN						:= FALSE;
			fbEcGetSlaveState.bExecute		:= TRUE;
			iState							:= iState + 10;
		END_IF
		
	30:																// Done already?
		fbEcGetSlaveState.bExecute			:= FALSE;	
		IF NOT fbEcGetSlaveState.bBusy THEN
			IF NOT fbEcGetSlaveState.bError AND fbEcGetSlaveState.state.deviceState = fbEcReqSlaveState.state THEN
				bBusy						:= FALSE;
				bDone						:= TRUE;
				iState						:= 0;
			ELSIF iTry = 40 THEN
				iState						:= 99;
			ELSE
				iTry						:= iTry + 1;
				iState						:= iState - 10;			
			END_IF
			byActualState					:= fbEcGetSlaveState.state.deviceState;
		END_IF
		
	99:																// ERROR STATE
		bError 								:= TRUE;
		bBusy								:= FALSE;
		udiErrorID							:= fbEcReqSlaveState.nErrId + fbEcGetSlaveState.nErrId;
		iState								:= 0;
		
END_CASE

fbEcReqSlaveState();
fbEcGetSlaveState();

END_FUNCTION_BLOCK

// ---- POUs/FB/POUsAxisOnline/AX5000/FB_HoldingBrakeCtrlAX5000.TcPOU
//==================================================================================================
//							Beckhoff Automation Poland
//									23.05.2018
//	Blok funkcyjny kontroli luzownika w silniku podpietym do AX5000. Przewaga ForceLock
//	Datatype:		ENUM (INT16)
//	Enum Value:		0 (0x00): 	Release_force
//					1 (0x01): 	Force_lock
//					2 (0x02): 	Force_unlock
//
// 	v1.1	|| TC v 3.1.4022.16	|| - optymalizacja kodu
//  v1.0	|| TC v 3.1.4022.16	|| - pierwsza wersja
//==================================================================================================
FUNCTION_BLOCK FB_HoldingBrakeCtrlAX5000
VAR_INPUT
	bForceLock 						: BOOL;								// 
	bForceUnlock					: BOOL;								// 
END_VAR
VAR_OUTPUT
	bBusy							: BOOL;
	bError							: BOOL; 							// General error: parameter or CoE read.
																		// If bError = TRUE and bInitialized = FALSE - error during read motor data.
																		// If bError = TRUE and bInitialized = TRUE and (iAdsErrId <> 0 or iCANopenErrId <> 0) then I2T read error
																		// If bError = TRUE and bInitialized = TRUE and iAdsErrId = 0 and iCANopenErrId = 0 then parameter error: rTorqueLimit outside permitted range rTorqueLimitLow..rTorqueLimitHigh or Empty stDriveRef
	iAdsErrId						: UINT;								// Forwarded output FB_SoEWrite
	iSecErrId						: UINT;								// Forwarded output FB_SoEWrite
END_VAR
VAR_IN_OUT
	Axis							: AXIS_REF;
END_VAR
VAR
	bExecute						: BOOL;
	iMotorBrakeForce				: INT;								// 0 - Release_force, 1 - Force_lock, 2 - Force_unlock
	fbSoEWrite						: FB_SoEWrite;
	rtForceLock						: R_TRIG;
	rtForceUnlock					: R_TRIG;
	ftForceLock						: F_TRIG;
	ftForceUnlock					: F_TRIG;
END_VAR

{region "Call triggers"}
//======================= Call triggers =========================
rtForceLock(CLK:= bForceLock);
ftForceLock(CLK:= bForceLock);
rtForceUnlock(CLK:= bForceUnlock);
ftForceUnlock(CLK:= bForceUnlock);
bExecute								:= rtForceLock.Q OR ftForceLock.Q OR rtForceUnlock.Q OR ftForceUnlock.Q;
//===============================================================
{endregion}
{region "Main code"}
//========================= Main code ===========================
IF bExecute THEN
	iMotorBrakeForce 						:= 0;										// Clear value
	iMotorBrakeForce.1 						:= bForceUnlock;							// Set force unlock bit
	iMotorBrakeForce 						:= SEL(bForceLock, iMotorBrakeForce, 1);	// Set force lock bit, it has higher priority than unlock
END_IF
	 
fbSoEWrite(
	NetId			:= '' , 
	Idn				:= P_0_IDN + 96 , 
	Element			:= 16#40 , 
	pSrcBuf			:= ADR(iMotorBrakeForce), 
	BufLen			:= SIZEOF(iMotorBrakeForce) , 
	Execute			:= bExecute , 
	Timeout			:= T#2S, 
	Axis			:= Axis , 
	Busy			=> bBusy , 
	Error			=> bError, 
	AdsErrId		=> iAdsErrId, 
	SercosErrId		=> iSecErrId );
//===============================================================
{endregion}

END_FUNCTION_BLOCK

// ---- POUs/FB/POUsAxisOnline/AX5000/FB_McAxisOnlineAX5000.TcPOU
//==================================================================================================
//							Beckhoff Automation Poland
//									7.12.2018
//	Wszystkomajacy blok funkcyjny do sterowania osia, 
//	wymagane biblioteki: Tc2_EtherCAT, Tc2_Drive, Tc2_MC2_Drive, Tc2_MC2, Tc2_Utilities
//  v1.2	|| TC v 3.1.4022.27		|| - dodane opisy bledow w formie zmiennych typu string
// 	v1.1 	|| TC v 3.1.4022.20	 	|| - ACT_MotorMonitoring - only for real axis
// 	v1.0 	|| TC v 3.1.4022.16	 	|| - first edition
//==================================================================================================
{attribute 'reflection'}
FUNCTION_BLOCK FB_McAxisOnlineAX5000
VAR_IN_OUT
	stMcAxisOnline						: ST_McAxisOnline;
	Axis								: AXIS_REF;
END_VAR
VAR
	mcPower								: MC_Power;
	mcStop								: MC_Stop;
	mcHalt								: MC_Halt;
	mcStopSS1							: MC_Stop;
	mcStopSS2							: MC_Stop;
	mcReset								: MC_Reset;
	mcHome								: MC_Home;
	mcSetPosition						: MC_SetPosition;
	fbSetPositionOffset					: FB_SetPositionOffset;
	mcJog								: MC_Jog;

	mcMoveAbsolute						: MC_MoveAbsolute;
	mcMoveRelative						: MC_MoveRelative;
	mcMoveVelocity						: MC_MoveVelocity;
	mcMoveModulo						: MC_MoveModulo;
	mcMoveAbsolute2						: MC_MoveAbsolute;
	mcMoveRelative2						: MC_MoveRelative;
	mcMoveVelocity2						: MC_MoveVelocity;
	mcMoveModulo2						: MC_MoveModulo;

	fbMotorMonitoring					: FB_MotorMonitoringAX5000;
	fbHoldingBrakeCtrl					: FB_HoldingBrakeCtrlAX5000;
	fbNcLimitSwitch						: FB_NcSWLimitSwitchCtrl;
	tonGetDriveDiag						: TON;
	fbReadChannelErrorCode				: FB_AxisDiag;
	
	mcReadDriveAddress					: MC_ReadDriveAddress;
	mcReadParameterSet					: MC_ReadParameterSet;
	fbGetDriveRef						: FB_GetDriveRef;

	// Internal
	bInitialized						: BOOL;
			
	// Initialization
	iInitStep							: INT;
	bInitializationError				: BOOL;
	wInitializationErrorCounter			: WORD;
	bDriveAddressReady					: BOOL;
	bDriveRefReady						: BOOL;
	bReadParameterSetReady				: BOOL;
	tonDelay							: TON;
	// Re init
	udiOnlineChangeCntOld				: UDINT;
	bOnlineChangeDetected				: BOOL;
	bReInit								: BOOL;
	bReInitialized						: BOOL;
	bReInitializationError				: BOOL;
	// Axis diag struct
	stAX5000Diag						: ST_AX5000Diag;
	{attribute 'instance-path'}
	{attribute 'noinit'}
	sInstancePath						: STRING;
END_VAR

// Device dependent initialization 
ACT_Initialization();
// Device independent commands, mostly NC 
ACT_States();
ACT_SWLimitSwitch();
ACT_Stop();
ACT_Power();
ACT_Homing();
ACT_Jog();
ACT_Move();
ACT_ResetAndDiag();
ACT_SetPosition();
// Device dependent commands
// Motor monitoring possible only with real axis
IF NOT Axis.Status.OpMode.SimulationAxis THEN
	ACT_MotorMonitoring();
END_IF
// Device dependent commands, possible only on real axis after complete initialization
IF bInitialized AND NOT Axis.Status.OpMode.SimulationAxis THEN
	ACT_SetPositionIO();
	ACT_HoldingBrakeCtrl();
END_IF

// Device independent error collection
ACT_ErrorCollection();

ACTION ACT_ErrorCollection:
// Error flags
stMcAxisOnline.stError.bDriveError					:= Axis.Status.DriveDeviceError;

stMcAxisOnline.stError.bNcError						:= Axis.Status.Error;

stMcAxisOnline.stError.bFBError						:= stMcAxisOnline.mcPower.bError OR stMcAxisOnline.mcReset.bError OR stMcAxisOnline.mcHome.bError OR stMcAxisOnline.mcJog.bError
													OR stMcAxisOnline.mcHalt.bError OR stMcAxisOnline.mcStop.bError OR stMcAxisOnline.mcSS1.bError OR stMcAxisOnline.mcSS2.bError
													OR stMcAxisOnline.mcMoveAbsolute.bError OR stMcAxisOnline.mcMoveRelative.bError OR stMcAxisOnline.mcMoveVelocity.bError OR stMcAxisOnline.mcMoveModulo.bError
													OR stMcAxisOnline.mcMoveAbsolute2.bError OR stMcAxisOnline.mcMoveRelative2.bError OR stMcAxisOnline.mcMoveVelocity2.bError OR stMcAxisOnline.mcMoveModulo2.bError
													OR stMcAxisOnline.stNcLimitSwitch.bError OR stMcAxisOnline.mcSetPosition.bError;
									
stMcAxisOnline.stError.bCommunicationError			:= stMcAxisOnline.stChannelErrorCode.bError OR stMcAxisOnline.stSetPositionOffset.bError OR stMcAxisOnline.stMotorMonitoring.bError OR stMcAxisOnline.stHoldingBrake.bError;

stMcAxisOnline.stError.bError						:= stMcAxisOnline.stError.bDriveError OR stMcAxisOnline.stError.bNcError OR stMcAxisOnline.stError.bFBError OR stMcAxisOnline.stError.bCommunicationError;
stMcAxisOnline.bError								:= stMcAxisOnline.stError.bError; // Forward one stage up

// Error codes
stMcAxisOnline.stError.uiDriveErrorID 				:= stMcAxisOnline.stChannelErrorCode.uiChannelErrorCode;
stMcAxisOnline.stError.uiDriveErrorIDHex 			:= stMcAxisOnline.stChannelErrorCode.uiChannelErrorCodeHex;

stMcAxisOnline.stError.udiNcErrorID 				:= Axis.Status.ErrorID;
stMcAxisOnline.stError.udiNcErrorIDHex 				:= Axis.Status.ErrorID;
	

stMcAxisOnline.stError.udiFBErrorID 				:= 	stMcAxisOnline.mcPower.udiErrorID + 
														stMcAxisOnline.mcReset.udiErrorID + 
														stMcAxisOnline.mcHome.udiErrorID + 
														stMcAxisOnline.mcJog.udiErrorID +
														stMcAxisOnline.mcHalt.udiErrorID + 
														stMcAxisOnline.mcStop.udiErrorID + 
														stMcAxisOnline.mcSS1.udiErrorID + 
														stMcAxisOnline.mcSS2.udiErrorID +
														stMcAxisOnline.mcMoveAbsolute.udiErrorID + 
														stMcAxisOnline.mcMoveRelative.udiErrorID + 
														stMcAxisOnline.mcMoveVelocity.udiErrorID + 
														stMcAxisOnline.mcMoveModulo.udiErrorID +
														stMcAxisOnline.mcMoveAbsolute2.udiErrorID + 
														stMcAxisOnline.mcMoveRelative2.udiErrorID + 
														stMcAxisOnline.mcMoveVelocity2.udiErrorID + 
														stMcAxisOnline.mcMoveModulo2.udiErrorID +
														stMcAxisOnline.stNcLimitSwitch.udiErrorID + 
														stMcAxisOnline.mcSetPosition.udiErrorID;

stMcAxisOnline.stError.udiFBErrorIDHex 				:= stMcAxisOnline.stError.udiFBErrorID;

stMcAxisOnline.stError.udiErrorID					:= stMcAxisOnline.stSetPositionOffset.udiErrorID;
stMcAxisOnline.stError.uiAdsErrorID					:= stMcAxisOnline.stChannelErrorCode.uiAdsErrId + stMcAxisOnline.stMotorMonitoring.uiAdsErrId + stMcAxisOnline.stHoldingBrake.uiAdsErrId;
stMcAxisOnline.stError.uiSecErrorID					:= stMcAxisOnline.stChannelErrorCode.uiSecErrId + stMcAxisOnline.stMotorMonitoring.uiSecErrId + stMcAxisOnline.stHoldingBrake.uiSecErrId;

stMcAxisOnline.stError.sNcError						:= F_AxErrMsg(stMcAxisOnline.stError.udiNcErrorID);
stMcAxisOnline.stError.sDriveError					:= F_AX5xErrMsg(stMcAxisOnline.stError.uiDriveErrorID);
END_ACTION

ACTION ACT_HoldingBrakeCtrl:
fbHoldingBrakeCtrl(
					bForceLock			:= stMcAxisOnline.stHoldingBrake.bForceLock,
					bForceUnlock		:= stMcAxisOnline.stHoldingBrake.bForceUnlock,
					bBusy				=> stMcAxisOnline.stHoldingBrake.bBusy,
					bError				=> stMcAxisOnline.stHoldingBrake.bError,
					iAdsErrId			=> stMcAxisOnline.stHoldingBrake.uiAdsErrId,
					iSecErrId			=>stMcAxisOnline.stHoldingBrake.uiSecErrId , 
					Axis				:= Axis );
END_ACTION

ACTION ACT_Homing:
mcHome(		Axis						:= Axis,
			Execute						:= stMcAxisOnline.mcHome.bExecute,
			Position					:= stMcAxisOnline.mcHome.lrPosition,
			HomingMode					:= stMcAxisOnline.mcHome.eHomingMode,
			BufferMode					:= stMcAxisOnline.mcHome.eBufferMode,
			Options						:= stMcAxisOnline.mcHome.stOptions,
			bCalibrationCam				:= stMcAxisOnline.mcHome.bCalibrationCam,
			Done						=> stMcAxisOnline.mcHome.bDone,
			Busy						=> stMcAxisOnline.mcHome.bBusy,
			Active						=> stMcAxisOnline.mcHome.bActive,
			CommandAborted				=> stMcAxisOnline.mcHome.bCommandAborted,
			Error						=> stMcAxisOnline.mcHome.bError,
			ErrorID						=> stMcAxisOnline.mcHome.udiErrorID);
END_ACTION

ACTION ACT_Initialization:
// bInitialized flag is set just once. 
// bReInitialized ise set each time we do online change or request reinit operation
// bDriveAddressReady, bReadParameterSetReady, bDriveRefReady - set just once after successed read

// Online change detection
bOnlineChangeDetected					:= udiOnlineChangeCntOld <> _AppInfo.OnlineChangeCnt;
udiOnlineChangeCntOld 					:= _AppInfo.OnlineChangeCnt;
// Reset init
IF bReInit OR bOnlineChangeDetected THEN
	iInitStep							:= 0;
END_IF

//Initialization process
CASE iInitStep OF
	0:	// Read Drive Address
		
		stMcAxisOnline.mcReadDriveAddress.bExecute	:=	 TRUE;
		iInitStep						:= iInitStep + 10;
		
	10: // Wait for data
	
		IF NOT stMcAxisOnline.mcReadDriveAddress.bBusy THEN
			stMcAxisOnline.mcReadDriveAddress.bExecute	:=	 FALSE;
			IF stMcAxisOnline.mcReadDriveAddress.bDone THEN
				iInitStep 				:= iInitStep + 10;
				bDriveAddressReady 		:= TRUE;
			ELSE
				iInitStep 				:= 1000;		// Error step
			END_IF
		END_IF
		
	20:	// Read Parameter Set
		
		stMcAxisOnline.mcReadParameterSet.bExecute		:=	 TRUE;
		iInitStep						:= iInitStep + 10;
		
	30: // Wait for data
	
		IF NOT stMcAxisOnline.mcReadParameterSet.bBusy THEN
			stMcAxisOnline.mcReadParameterSet.bExecute	:=	 FALSE;
			IF stMcAxisOnline.mcReadParameterSet.bDone THEN
				iInitStep 				:= iInitStep + 10;
				bReadParameterSetReady 	:= TRUE;
			ELSE
				iInitStep 				:= 1000;		// Error step
			END_IF
		END_IF	
	
	40:	// Get Drive Ref
		
		stMcAxisOnline.stGetDriveRef.bExecute		:=	 TRUE;
		iInitStep						:= iInitStep + 10;
		
	50: // Wait for data
	
		IF NOT stMcAxisOnline.stGetDriveRef.bBusy THEN
			stMcAxisOnline.stGetDriveRef.bExecute	:=	 FALSE;
			IF NOT stMcAxisOnline.stGetDriveRef.bError THEN
				iInitStep 				:= iInitStep + 10;
				bDriveRefReady 			:= TRUE;
			ELSE
				iInitStep 				:= 1000;		// Error step
			END_IF
		END_IF
	
	60: // Success - initialized flag, clear error
		bReInitialized					:= bInitialized;	// TRUE only when it's not first initialization e.g. online change
		bInitialized 					:= TRUE;
		bReInitializationError			:= FALSE;			// TRUE only when it's not first initialization e.g. online change
		bInitializationError			:= FALSE;
		iInitStep 						:= iInitStep + 10;
		
	70: // Idle
	
		;
		
	1000: // Error step
		wInitializationErrorCounter 	:= wInitializationErrorCounter + 1;
		IF wInitializationErrorCounter < 100 THEN
			iInitStep					:= iInitStep + 5;			// Go to delay
		ELSE
			bReInitializationError		:= bInitializationError;	// TRUE only when it's not first initialization e.g. online change
			bInitializationError		:= TRUE;
			bReInitialized				:= FALSE;
			iInitStep 					:= iInitStep + 10;
		END_IF

	1005: // Delay step
		tonDelay(IN:= TRUE, PT:= T#1S);
		IF tonDelay.Q THEN
			tonDelay(IN:= FALSE, PT:= T#1S);
			iInitStep					:= 0;
		END_IF
		
	1010: // Idle after error
		;
	
END_CASE

mcReadDriveAddress(	Axis				:= Axis,
					Execute				:= stMcAxisOnline.mcReadDriveAddress.bExecute,
					Done				=> stMcAxisOnline.mcReadDriveAddress.bDone,
					Busy				=> stMcAxisOnline.mcReadDriveAddress.bBusy,
					Error				=> stMcAxisOnline.mcReadDriveAddress.bError,
					ErrorID				=> stMcAxisOnline.mcReadDriveAddress.udiErrorID,
					DriveAddress		=> stMcAxisOnline.stDriveAddress);
				
mcReadParameterSet(	Parameter			:= stMcAxisOnline.stAxisParameter,
					Axis				:= Axis,
					Execute				:= stMcAxisOnline.mcReadParameterSet.bExecute,
					Done				=> stMcAxisOnline.mcReadParameterSet.bDone,
					Busy				=> stMcAxisOnline.mcReadParameterSet.bBusy,
					Error				=> stMcAxisOnline.mcReadParameterSet.bError,
					ErrorID				=> stMcAxisOnline.mcReadParameterSet.udiErrorID);
					
fbGetDriveRef(		bExecute			:= stMcAxisOnline.stGetDriveRef.bExecute,
					bBusy				=> stMcAxisOnline.stGetDriveRef.bBusy,
					bError				=> stMcAxisOnline.stGetDriveRef.bError,
					udiErrorID			=> stMcAxisOnline.stGetDriveRef.udiErrorID,
					stDriveRef			=> stMcAxisOnline.stDriveRef,
					Axis				:= Axis);
END_ACTION

ACTION ACT_Jog:
// Direct access from bSlow or bFast, if none then free choice
IF stMcAxisOnline.mcJog.bSlowForward OR stMcAxisOnline.mcJog.bSlowBackward THEN
	stMcAxisOnline.mcJog.eMode			:= MC_JOGMODE_STANDARD_SLOW;
ELSIF stMcAxisOnline.mcJog.bFastForward OR stMcAxisOnline.mcJog.bFastBackward THEN
	stMcAxisOnline.mcJog.eMode			:= MC_JOGMODE_STANDARD_FAST;
END_IF

mcJog(		Axis						:= Axis,
			JogForward					:= stMcAxisOnline.mcJog.bJogForward OR stMcAxisOnline.mcJog.bSlowForward OR stMcAxisOnline.mcJog.bFastForward,
			JogBackwards				:= stMcAxisOnline.mcJog.bJogBackwards OR stMcAxisOnline.mcJog.bSlowBackward OR stMcAxisOnline.mcJog.bFastBackward,
			Mode						:= stMcAxisOnline.mcJog.eMode,
			Position					:= stMcAxisOnline.mcJog.lrPosition,
			Velocity					:= stMcAxisOnline.mcJog.lrVelocity,
			Acceleration				:= stMcAxisOnline.mcJog.lrAcceleration,
			Deceleration				:= stMcAxisOnline.mcJog.lrDeceleration,
			Jerk						:= stMcAxisOnline.mcJog.lrJerk,
			Done						=> stMcAxisOnline.mcJog.bDone,
			Busy						=> stMcAxisOnline.mcJog.bBusy,
			Active						=> stMcAxisOnline.mcJog.bActive,
			CommandAborted				=> stMcAxisOnline.mcJog.bCommandAborted,
			Error						=> stMcAxisOnline.mcJog.bError,
			ErrorID						=> stMcAxisOnline.mcJog.udiErrorID);
END_ACTION

ACTION ACT_MotorMonitoring:
fbMotorMonitoring(
					bReset				:= stMcAxisOnline.stMotorMonitoring.bReset, 
					rTorqueLimit		:= stMcAxisOnline.stMotorMonitoring.rTorqueLimit , 
					bError				=> stMcAxisOnline.stMotorMonitoring.bError , 
					uiAdsErrId			=> stMcAxisOnline.stMotorMonitoring.uiAdsErrId , 
					uiSercosErrId		=> stMcAxisOnline.stMotorMonitoring.uiSecErrId, 
					bInitialized		=> stMcAxisOnline.stMotorMonitoring.bInitialized , 
					bWarning			=> stMcAxisOnline.stMotorMonitoring.bWarning , 
					rWarningCurrent		=> stMcAxisOnline.stMotorMonitoring.rWarningCurrent , 
					rTorquePerc			=> stMcAxisOnline.stMotorMonitoring.rTorquePerc,
					rTorquePercMax		=> stMcAxisOnline.stMotorMonitoring.rTorquePercMax,
					rTorque				=> stMcAxisOnline.stMotorMonitoring.rTorque , 
					rTorqueF			=> stMcAxisOnline.stMotorMonitoring.rTorqueF , 
					rTorqueMax			=> stMcAxisOnline.stMotorMonitoring.rTorqueMax , 
					rCurrent			=> stMcAxisOnline.stMotorMonitoring.rCurrent , 
					rCurrentF			=> stMcAxisOnline.stMotorMonitoring.rCurrentF , 
					rCurrentMax			=> stMcAxisOnline.stMotorMonitoring.rCurrentMax , 
					rI2T				=> stMcAxisOnline.stMotorMonitoring.rI2T , 
					rI2TMax				=> stMcAxisOnline.stMotorMonitoring.rI2TMax , 
					Axis				:= Axis );
END_ACTION

